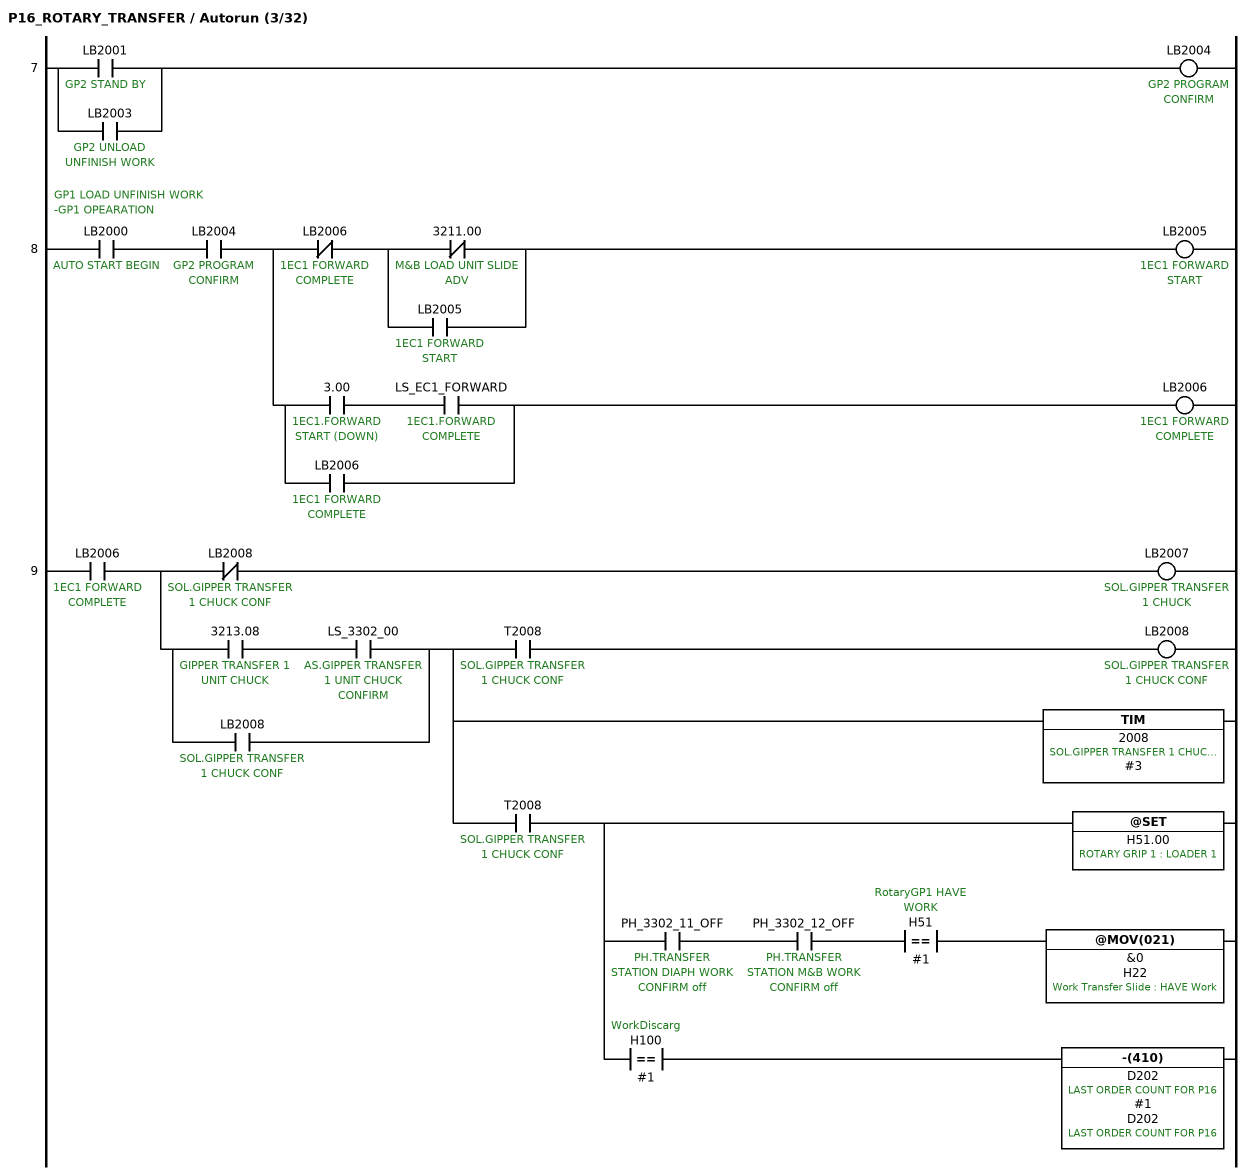
; [picture p240: P16_ROTARY_TRANSFER / Autorun, rungs 7-9]
; rung 7
LD LB2001  ; GP2 STAND BY
OR LB2003  ; GP2 UNLOAD UNFINISH WORK
OUT LB2004  ; GP2 PROGRAM CONFIRM
; rung 8: GP1 LOAD UNFINISH WORK / -GP1 OPEARATION
LD LB2000  ; AUTO START BEGIN
AND LB2004  ; GP2 PROGRAM CONFIRM
OUT TR0
ANDNOT LB2006  ; 1EC1 FORWARD COMPLETE
LDNOT 3211.00  ; M&B LOAD UNIT SLIDE ADV
OR LB2005  ; 1EC1 FORWARD START
ANDLD
OUT LB2005  ; 1EC1 FORWARD START
LD TR0
LD 3.00  ; 1EC1.FORWARD START (DOWN)
AND LS_EC1_FORWARD  ; 1EC1.FORWARD COMPLETE
OR LB2006  ; 1EC1 FORWARD COMPLETE
ANDLD
OUT LB2006  ; 1EC1 FORWARD COMPLETE
; rung 9
LD LB2006  ; 1EC1 FORWARD COMPLETE
OUT TR0
ANDNOT LB2008  ; SOL.GIPPER TRANSFER 1 CHUCK CONF
OUT LB2007  ; SOL.GIPPER TRANSFER 1 CHUCK
LD TR0
LD 3213.08  ; GIPPER TRANSFER 1 UNIT CHUCK
AND LS_3302_00  ; AS.GIPPER TRANSFER 1 UNIT CHUCK CONFIRM
OR LB2008  ; SOL.GIPPER TRANSFER 1 CHUCK CONF
ANDLD
OUT TR0
AND T2008  ; SOL.GIPPER TRANSFER 1 CHUCK CONF
OUT LB2008  ; SOL.GIPPER TRANSFER 1 CHUCK CONF
LD TR0
TIM 2008 #3  ; SOL.GIPPER TRANSFER 1 CHUCK CONF
AND T2008  ; SOL.GIPPER TRANSFER 1 CHUCK CONF
OUT TR0
@SET H51.00  ; ROTARY GRIP 1 : LOADER 1
AND PH_3302_11_OFF  ; PH.TRANSFER STATION DIAPH WORK CONFIRM off
AND PH_3302_12_OFF  ; PH.TRANSFER STATION M&B WORK CONFIRM off
AND=(300) H51 #1  ; RotaryGP1 HAVE WORK
@MOV(021) &0 H22  ; Work Transfer Slide : HAVE Work
LD TR0
AND=(300) H100 #1  ; WorkDiscarg
-(410) D202 #1 D202  ; LAST ORDER COUNT FOR P16

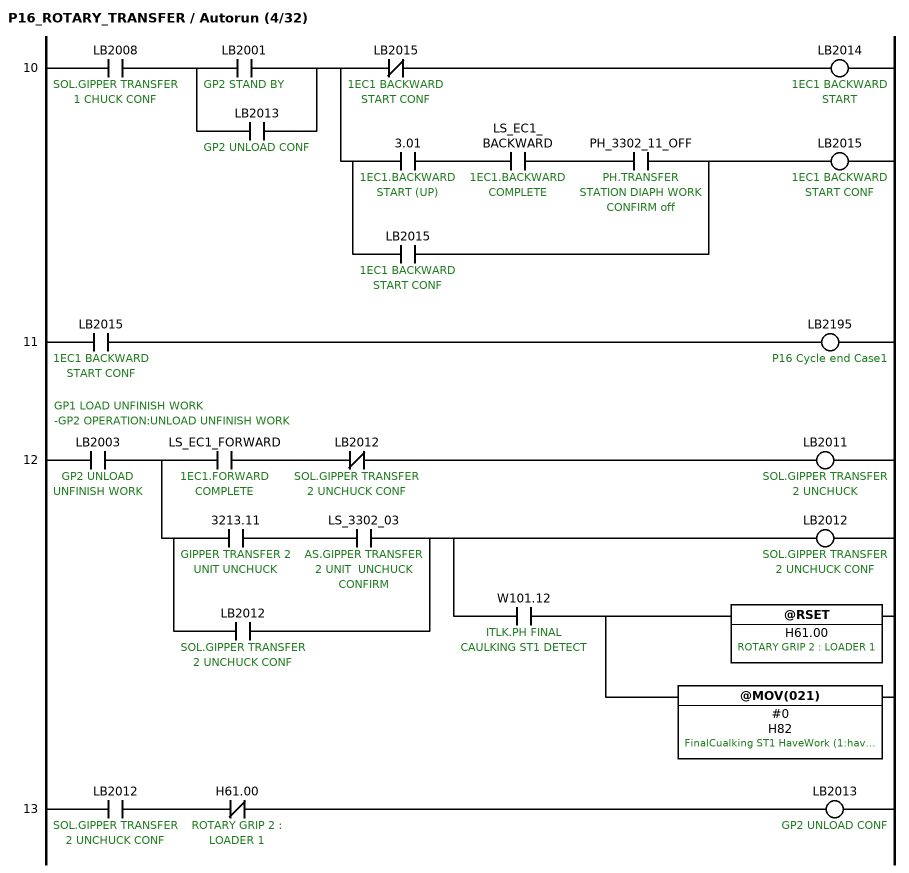
; rung 10
LD LB2008  ; SOL.GIPPER TRANSFER 1 CHUCK CONF
LD LB2001  ; GP2 STAND BY
OR LB2013  ; GP2 UNLOAD CONF
ANDLD
OUT TR0
ANDNOT LB2015  ; 1EC1 BACKWARD START CONF
OUT LB2014  ; 1EC1 BACKWARD START
LD TR0
LD 3.01  ; 1EC1.BACKWARD START (UP)
AND LS_EC1_BACKWARD  ; 1EC1.BACKWARD COMPLETE
AND PH_3302_11_OFF  ; PH.TRANSFER STATION DIAPH WORK CONFIRM off
OR LB2015  ; 1EC1 BACKWARD START CONF
ANDLD
OUT LB2015  ; 1EC1 BACKWARD START CONF
; rung 11
LD LB2015  ; 1EC1 BACKWARD START CONF
OUT LB2195  ; P16 Cycle end Case1
; rung 12: GP1 LOAD UNFINISH WORK / -GP2 OPERATION:UNLOAD UNFINISH WORK
LD LB2003  ; GP2 UNLOAD UNFINISH WORK
OUT TR0
AND LS_EC1_FORWARD  ; 1EC1.FORWARD COMPLETE
ANDNOT LB2012  ; SOL.GIPPER TRANSFER 2 UNCHUCK CONF
OUT LB2011  ; SOL.GIPPER TRANSFER 2 UNCHUCK
LD TR0
LD 3213.11  ; GIPPER TRANSFER 2 UNIT UNCHUCK
AND LS_3302_03  ; AS.GIPPER TRANSFER 2 UNIT  UNCHUCK CONFIRM
OR LB2012  ; SOL.GIPPER TRANSFER 2 UNCHUCK CONF
ANDLD
OUT LB2012  ; SOL.GIPPER TRANSFER 2 UNCHUCK CONF
AND W101.12  ; ITLK.PH FINAL CAULKING ST1 DETECT
@RSET H61.00  ; ROTARY GRIP 2 : LOADER 1
@MOV(021) #0 H82  ; FinalCualking ST1 HaveWork (1:have work 2:no work)
; rung 13
LD LB2012  ; SOL.GIPPER TRANSFER 2 UNCHUCK CONF
ANDNOT H61.00  ; ROTARY GRIP 2 : LOADER 1
OUT LB2013  ; GP2 UNLOAD CONF

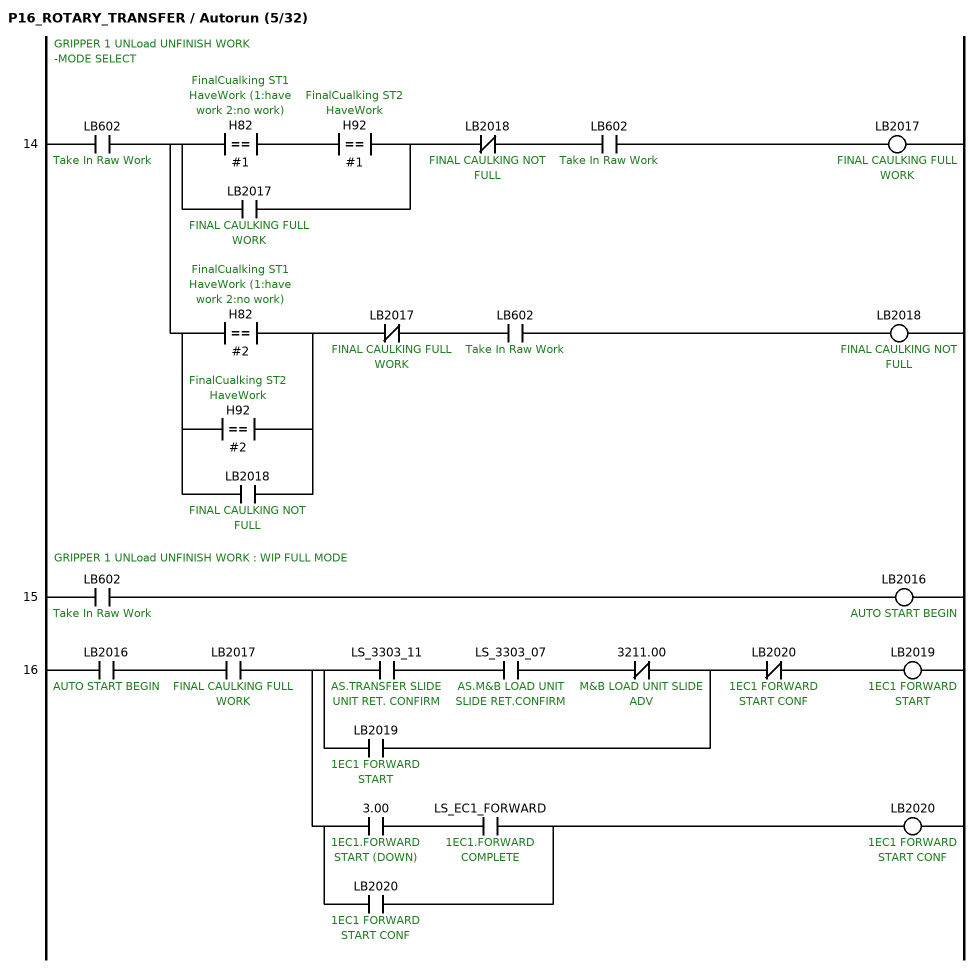
; rung 14: GRIPPER 1 UNLoad UNFINISH WORK / -MODE SELECT
LD LB602  ; Take In Raw Work
OUT TR0
LD=(300) H82 #1  ; FinalCualking ST1 HaveWork (1:have work 2:no work)
AND=(300) H92 #1  ; FinalCualking ST2 HaveWork
OR LB2017  ; FINAL CAULKING FULL WORK
ANDLD
ANDNOT LB2018  ; FINAL CAULKING NOT FULL
AND LB602  ; Take In Raw Work
OUT LB2017  ; FINAL CAULKING FULL WORK
LD TR0
LD=(300) H82 #2  ; FinalCualking ST1 HaveWork (1:have work 2:no work)
OR=(300) H92 #2  ; FinalCualking ST2 HaveWork
OR LB2018  ; FINAL CAULKING NOT FULL
ANDLD
ANDNOT LB2017  ; FINAL CAULKING FULL WORK
AND LB602  ; Take In Raw Work
OUT LB2018  ; FINAL CAULKING NOT FULL
; rung 15: GRIPPER 1 UNLoad UNFINISH WORK : WIP FULL MODE
LD LB602  ; Take In Raw Work
OUT LB2016  ; AUTO START BEGIN
; rung 16
LD LB2016  ; AUTO START BEGIN
AND LB2017  ; FINAL CAULKING FULL WORK
OUT TR0
LD LS_3303_11  ; AS.TRANSFER SLIDE UNIT RET. CONFIRM
AND LS_3303_07  ; AS.M&B LOAD UNIT SLIDE RET.CONFIRM
ANDNOT 3211.00  ; M&B LOAD UNIT SLIDE ADV
OR LB2019  ; 1EC1 FORWARD START
ANDLD
ANDNOT LB2020  ; 1EC1 FORWARD START CONF
OUT LB2019  ; 1EC1 FORWARD START
LD TR0
LD 3.00  ; 1EC1.FORWARD START (DOWN)
AND LS_EC1_FORWARD  ; 1EC1.FORWARD COMPLETE
OR LB2020  ; 1EC1 FORWARD START CONF
ANDLD
OUT LB2020  ; 1EC1 FORWARD START CONF

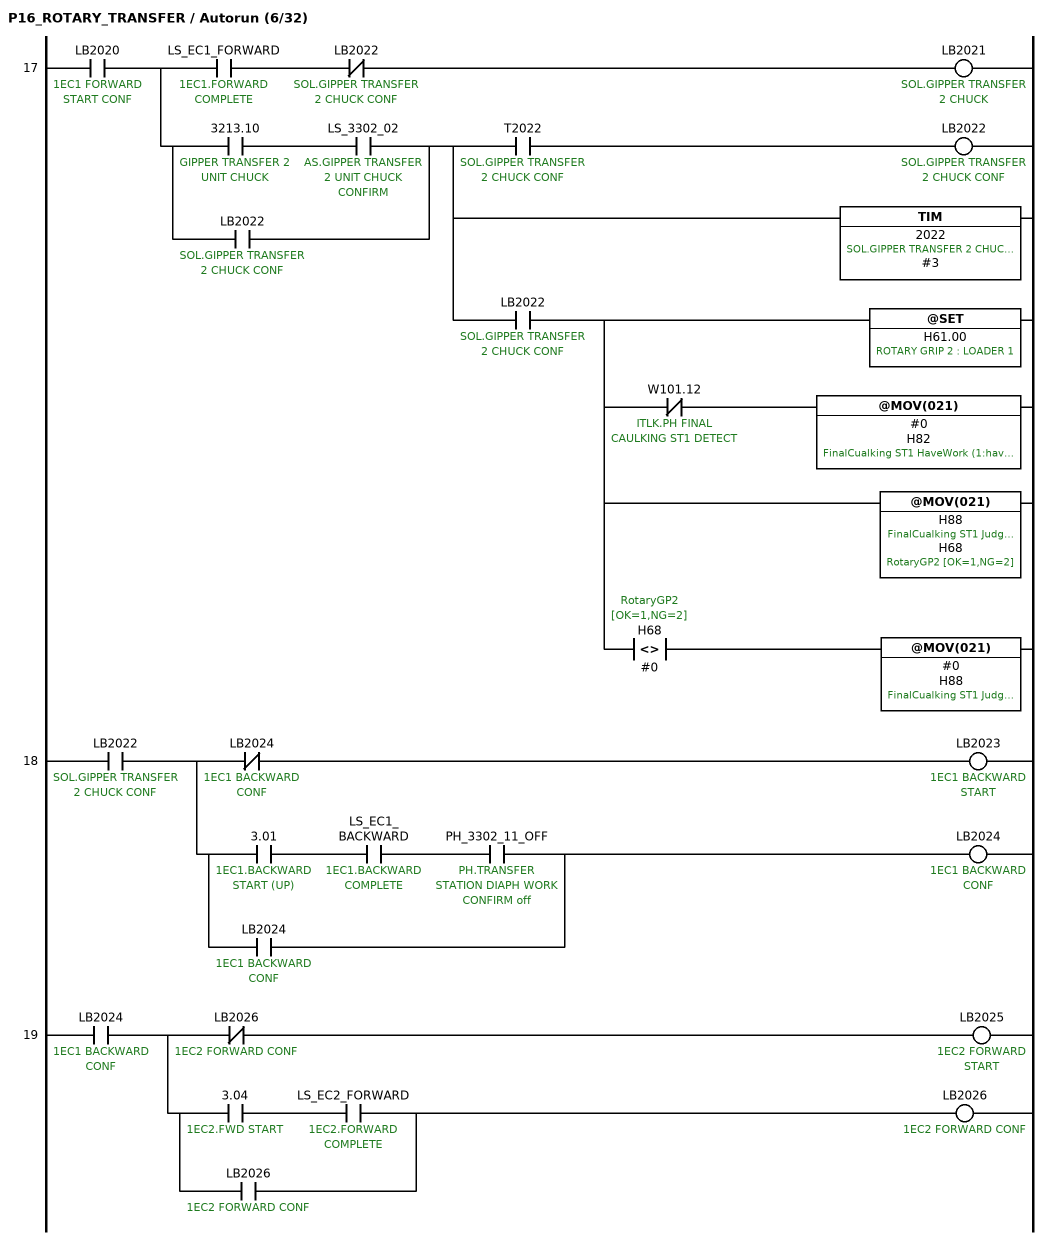
; rung 17
LD LB2020  ; 1EC1 FORWARD START CONF
OUT TR0
AND LS_EC1_FORWARD  ; 1EC1.FORWARD COMPLETE
ANDNOT LB2022  ; SOL.GIPPER TRANSFER 2 CHUCK CONF
OUT LB2021  ; SOL.GIPPER TRANSFER 2 CHUCK
LD TR0
LD 3213.10  ; GIPPER TRANSFER 2 UNIT CHUCK
AND LS_3302_02  ; AS.GIPPER TRANSFER 2 UNIT CHUCK CONFIRM
OR LB2022  ; SOL.GIPPER TRANSFER 2 CHUCK CONF
ANDLD
OUT TR0
AND T2022  ; SOL.GIPPER TRANSFER 2 CHUCK CONF
OUT LB2022  ; SOL.GIPPER TRANSFER 2 CHUCK CONF
LD TR0
TIM 2022 #3  ; SOL.GIPPER TRANSFER 2 CHUCK CONF
AND LB2022  ; SOL.GIPPER TRANSFER 2 CHUCK CONF
OUT TR0
@SET H61.00  ; ROTARY GRIP 2 : LOADER 1
ANDNOT W101.12  ; ITLK.PH FINAL CAULKING ST1 DETECT
@MOV(021) #0 H82  ; FinalCualking ST1 HaveWork (1:have work 2:no work)
LD TR0
@MOV(021) H88 H68  ; FinalCualking ST1 Judge [OK=1,NG=2], RotaryGP2 [OK=1,NG=2]
AND<>(305) H68 #0  ; RotaryGP2 [OK=1,NG=2]
@MOV(021) #0 H88  ; FinalCualking ST1 Judge [OK=1,NG=2]
; rung 18
LD LB2022  ; SOL.GIPPER TRANSFER 2 CHUCK CONF
OUT TR0
ANDNOT LB2024  ; 1EC1 BACKWARD CONF
OUT LB2023  ; 1EC1 BACKWARD START
LD TR0
LD 3.01  ; 1EC1.BACKWARD START (UP)
AND LS_EC1_BACKWARD  ; 1EC1.BACKWARD COMPLETE
AND PH_3302_11_OFF  ; PH.TRANSFER STATION DIAPH WORK CONFIRM off
OR LB2024  ; 1EC1 BACKWARD CONF
ANDLD
OUT LB2024  ; 1EC1 BACKWARD CONF
; rung 19
LD LB2024  ; 1EC1 BACKWARD CONF
OUT TR0
ANDNOT LB2026  ; 1EC2 FORWARD CONF
OUT LB2025  ; 1EC2 FORWARD START
LD TR0
LD 3.04  ; 1EC2.FWD START
AND LS_EC2_FORWARD  ; 1EC2.FORWARD COMPLETE
OR LB2026  ; 1EC2 FORWARD CONF
ANDLD
OUT LB2026  ; 1EC2 FORWARD CONF

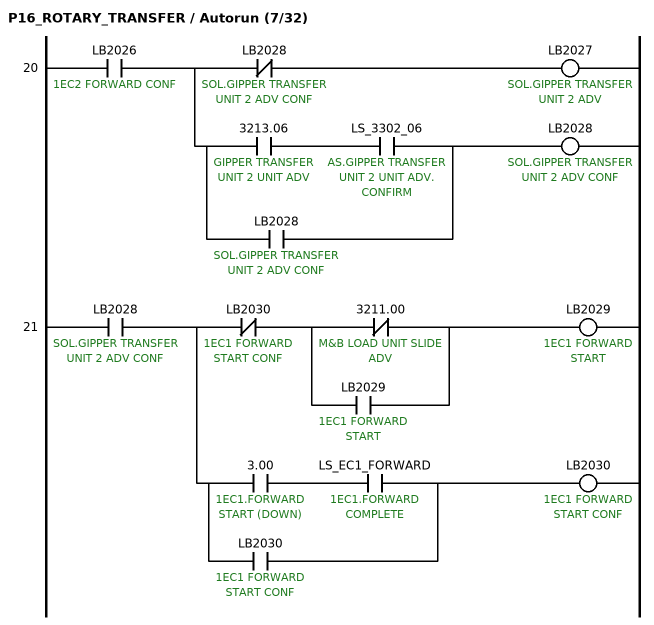
; rung 20
LD LB2026  ; 1EC2 FORWARD CONF
OUT TR0
ANDNOT LB2028  ; SOL.GIPPER TRANSFER UNIT 2 ADV CONF
OUT LB2027  ; SOL.GIPPER TRANSFER UNIT 2 ADV
LD TR0
LD 3213.06  ; GIPPER TRANSFER UNIT 2 UNIT ADV
AND LS_3302_06  ; AS.GIPPER TRANSFER UNIT 2 UNIT ADV. CONFIRM
OR LB2028  ; SOL.GIPPER TRANSFER UNIT 2 ADV CONF
ANDLD
OUT LB2028  ; SOL.GIPPER TRANSFER UNIT 2 ADV CONF
; rung 21
LD LB2028  ; SOL.GIPPER TRANSFER UNIT 2 ADV CONF
OUT TR0
ANDNOT LB2030  ; 1EC1 FORWARD START CONF
LDNOT 3211.00  ; M&B LOAD UNIT SLIDE ADV
OR LB2029  ; 1EC1 FORWARD START
ANDLD
OUT LB2029  ; 1EC1 FORWARD START
LD TR0
LD 3.00  ; 1EC1.FORWARD START (DOWN)
AND LS_EC1_FORWARD  ; 1EC1.FORWARD COMPLETE
OR LB2030  ; 1EC1 FORWARD START CONF
ANDLD
OUT LB2030  ; 1EC1 FORWARD START CONF

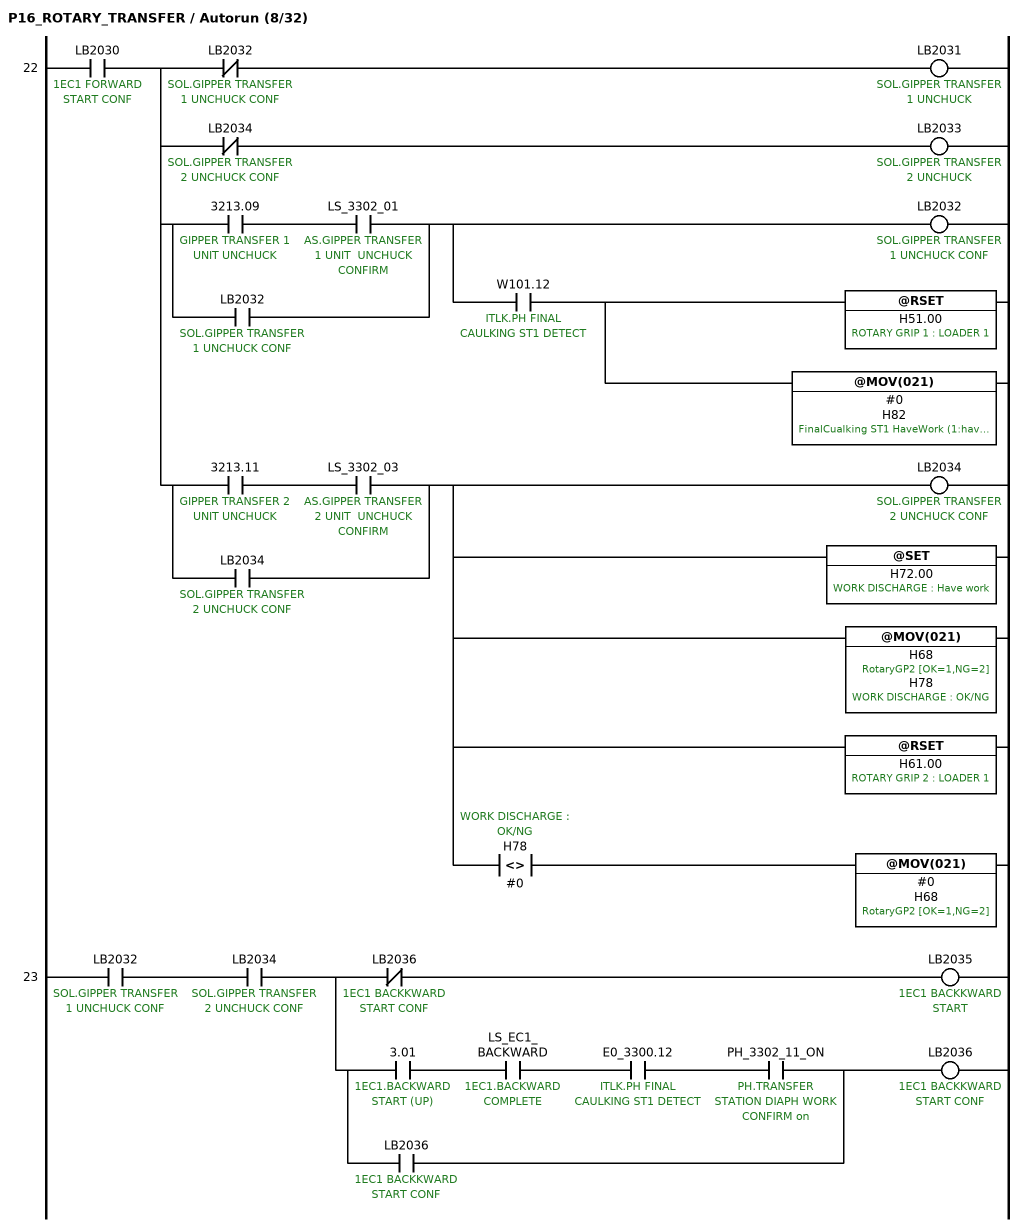
; rung 22
LD LB2030  ; 1EC1 FORWARD START CONF
OUT TR0
ANDNOT LB2032  ; SOL.GIPPER TRANSFER 1 UNCHUCK CONF
OUT LB2031  ; SOL.GIPPER TRANSFER 1 UNCHUCK
LD TR0
ANDNOT LB2034  ; SOL.GIPPER TRANSFER 2 UNCHUCK CONF
OUT LB2033  ; SOL.GIPPER TRANSFER 2 UNCHUCK
LD TR0
LD 3213.09  ; GIPPER TRANSFER 1 UNIT UNCHUCK
AND LS_3302_01  ; AS.GIPPER TRANSFER 1 UNIT  UNCHUCK CONFIRM
OR LB2032  ; SOL.GIPPER TRANSFER 1 UNCHUCK CONF
ANDLD
OUT LB2032  ; SOL.GIPPER TRANSFER 1 UNCHUCK CONF
AND W101.12  ; ITLK.PH FINAL CAULKING ST1 DETECT
@RSET H51.00  ; ROTARY GRIP 1 : LOADER 1
@MOV(021) #0 H82  ; FinalCualking ST1 HaveWork (1:have work 2:no work)
LD TR0
LD 3213.11  ; GIPPER TRANSFER 2 UNIT UNCHUCK
AND LS_3302_03  ; AS.GIPPER TRANSFER 2 UNIT  UNCHUCK CONFIRM
OR LB2034  ; SOL.GIPPER TRANSFER 2 UNCHUCK CONF
ANDLD
OUT LB2034  ; SOL.GIPPER TRANSFER 2 UNCHUCK CONF
@SET H72.00  ; WORK DISCHARGE : Have work
@MOV(021) H68 H78  ; RotaryGP2 [OK=1,NG=2], WORK DISCHARGE : OK/NG
@RSET H61.00  ; ROTARY GRIP 2 : LOADER 1
AND<>(305) H78 #0  ; WORK DISCHARGE : OK/NG
@MOV(021) #0 H68  ; RotaryGP2 [OK=1,NG=2]
; rung 23
LD LB2032  ; SOL.GIPPER TRANSFER 1 UNCHUCK CONF
AND LB2034  ; SOL.GIPPER TRANSFER 2 UNCHUCK CONF
OUT TR0
ANDNOT LB2036  ; 1EC1 BACKKWARD START CONF
OUT LB2035  ; 1EC1 BACKKWARD START
LD TR0
LD 3.01  ; 1EC1.BACKWARD START (UP)
AND LS_EC1_BACKWARD  ; 1EC1.BACKWARD COMPLETE
AND E0_3300.12  ; ITLK.PH FINAL CAULKING ST1 DETECT
AND PH_3302_11_ON  ; PH.TRANSFER STATION DIAPH WORK CONFIRM on
OR LB2036  ; 1EC1 BACKKWARD START CONF
ANDLD
OUT LB2036  ; 1EC1 BACKKWARD START CONF

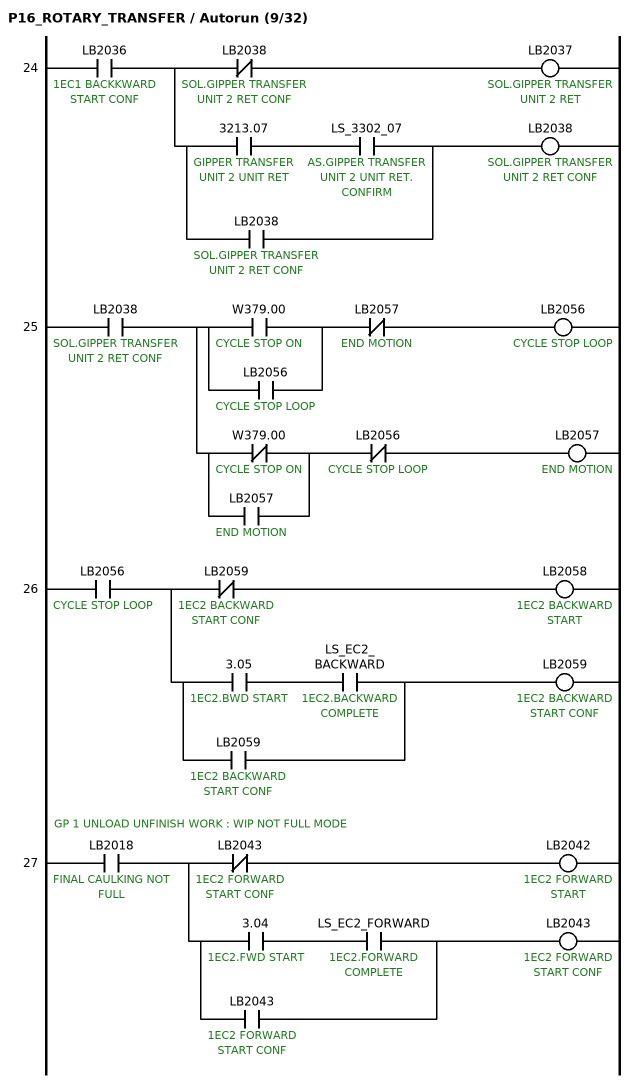
; rung 24
LD LB2036  ; 1EC1 BACKKWARD START CONF
OUT TR0
ANDNOT LB2038  ; SOL.GIPPER TRANSFER UNIT 2 RET CONF
OUT LB2037  ; SOL.GIPPER TRANSFER UNIT 2 RET
LD TR0
LD 3213.07  ; GIPPER TRANSFER UNIT 2 UNIT RET
AND LS_3302_07  ; AS.GIPPER TRANSFER UNIT 2 UNIT RET. CONFIRM
OR LB2038  ; SOL.GIPPER TRANSFER UNIT 2 RET CONF
ANDLD
OUT LB2038  ; SOL.GIPPER TRANSFER UNIT 2 RET CONF
; rung 25
LD LB2038  ; SOL.GIPPER TRANSFER UNIT 2 RET CONF
OUT TR0
LD W379.00  ; CYCLE STOP ON
OR LB2056  ; CYCLE STOP LOOP
ANDLD
ANDNOT LB2057  ; END MOTION
OUT LB2056  ; CYCLE STOP LOOP
LD TR0
LDNOT W379.00  ; CYCLE STOP ON
OR LB2057  ; END MOTION
ANDLD
ANDNOT LB2056  ; CYCLE STOP LOOP
OUT LB2057  ; END MOTION
; rung 26
LD LB2056  ; CYCLE STOP LOOP
OUT TR0
ANDNOT LB2059  ; 1EC2 BACKWARD START CONF
OUT LB2058  ; 1EC2 BACKWARD START
LD TR0
LD 3.05  ; 1EC2.BWD START
AND LS_EC2_BACKWARD  ; 1EC2.BACKWARD COMPLETE
OR LB2059  ; 1EC2 BACKWARD START CONF
ANDLD
OUT LB2059  ; 1EC2 BACKWARD START CONF
; rung 27: GP 1 UNLOAD UNFINISH WORK : WIP NOT FULL MODE
LD LB2018  ; FINAL CAULKING NOT FULL
OUT TR0
ANDNOT LB2043  ; 1EC2 FORWARD START CONF
OUT LB2042  ; 1EC2 FORWARD START
LD TR0
LD 3.04  ; 1EC2.FWD START
AND LS_EC2_FORWARD  ; 1EC2.FORWARD COMPLETE
OR LB2043  ; 1EC2 FORWARD START CONF
ANDLD
OUT LB2043  ; 1EC2 FORWARD START CONF

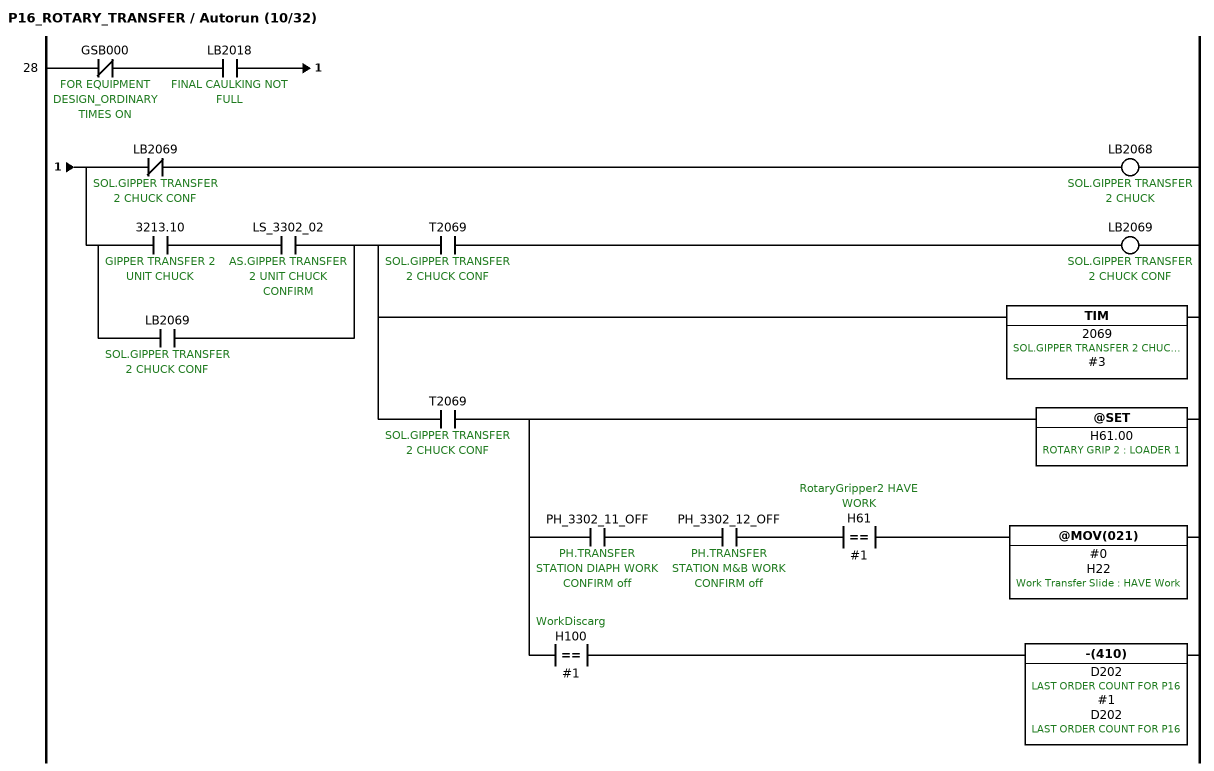
; rung 28
LDNOT GSB000  ; FOR EQUIPMENT DESIGN_ORDINARY TIMES ON
AND LB2018  ; FINAL CAULKING NOT FULL
OUT TR0
ANDNOT LB2069  ; SOL.GIPPER TRANSFER 2 CHUCK CONF
OUT LB2068  ; SOL.GIPPER TRANSFER 2 CHUCK
LD TR0
LD 3213.10  ; GIPPER TRANSFER 2 UNIT CHUCK
AND LS_3302_02  ; AS.GIPPER TRANSFER 2 UNIT CHUCK CONFIRM
OR LB2069  ; SOL.GIPPER TRANSFER 2 CHUCK CONF
ANDLD
OUT TR0
AND T2069  ; SOL.GIPPER TRANSFER 2 CHUCK CONF
OUT LB2069  ; SOL.GIPPER TRANSFER 2 CHUCK CONF
LD TR0
TIM 2069 #3  ; SOL.GIPPER TRANSFER 2 CHUCK CONF
AND T2069  ; SOL.GIPPER TRANSFER 2 CHUCK CONF
OUT TR0
@SET H61.00  ; ROTARY GRIP 2 : LOADER 1
AND PH_3302_11_OFF  ; PH.TRANSFER STATION DIAPH WORK CONFIRM off
AND PH_3302_12_OFF  ; PH.TRANSFER STATION M&B WORK CONFIRM off
AND=(300) H61 #1  ; RotaryGripper2 HAVE WORK
@MOV(021) #0 H22  ; Work Transfer Slide : HAVE Work
LD TR0
AND=(300) H100 #1  ; WorkDiscarg
-(410) D202 #1 D202  ; LAST ORDER COUNT FOR P16

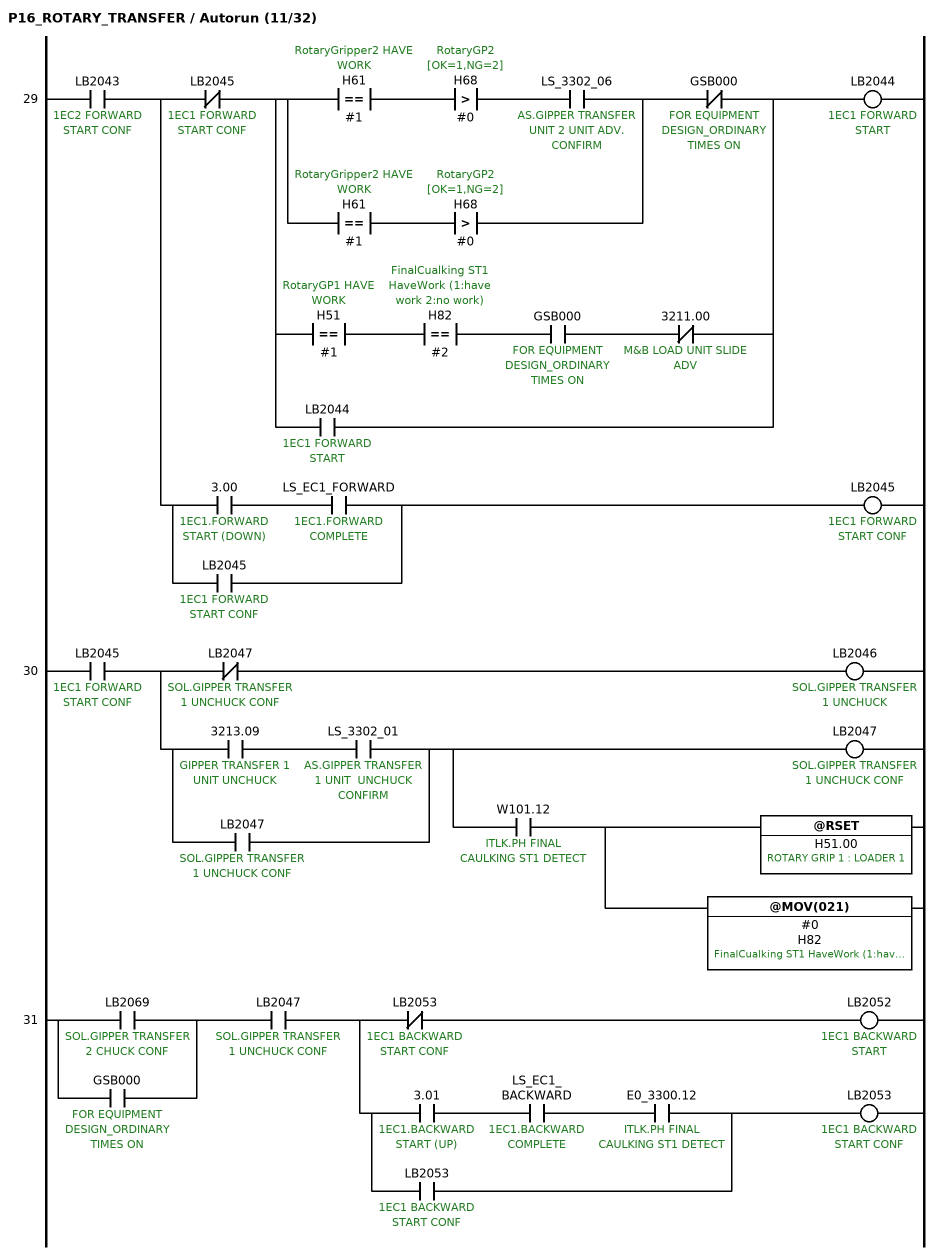
; rung 29
LD LB2043  ; 1EC2 FORWARD START CONF
OUT TR0
ANDNOT LB2045  ; 1EC1 FORWARD START CONF
LD=(300) H61 #1  ; RotaryGripper2 HAVE WORK
AND>(320) H68 #0  ; RotaryGP2 [OK=1,NG=2]
AND LS_3302_06  ; AS.GIPPER TRANSFER UNIT 2 UNIT ADV. CONFIRM
LD=(300) H61 #1  ; RotaryGripper2 HAVE WORK
AND>(320) H68 #0  ; RotaryGP2 [OK=1,NG=2]
ORLD
ANDNOT GSB000  ; FOR EQUIPMENT DESIGN_ORDINARY TIMES ON
LD=(300) H51 #1  ; RotaryGP1 HAVE WORK
AND=(300) H82 #2  ; FinalCualking ST1 HaveWork (1:have work 2:no work)
AND GSB000  ; FOR EQUIPMENT DESIGN_ORDINARY TIMES ON
ANDNOT 3211.00  ; M&B LOAD UNIT SLIDE ADV
ORLD
OR LB2044  ; 1EC1 FORWARD START
ANDLD
OUT LB2044  ; 1EC1 FORWARD START
LD TR0
LD 3.00  ; 1EC1.FORWARD START (DOWN)
AND LS_EC1_FORWARD  ; 1EC1.FORWARD COMPLETE
OR LB2045  ; 1EC1 FORWARD START CONF
ANDLD
OUT LB2045  ; 1EC1 FORWARD START CONF
; rung 30
LD LB2045  ; 1EC1 FORWARD START CONF
OUT TR0
ANDNOT LB2047  ; SOL.GIPPER TRANSFER 1 UNCHUCK CONF
OUT LB2046  ; SOL.GIPPER TRANSFER 1 UNCHUCK
LD TR0
LD 3213.09  ; GIPPER TRANSFER 1 UNIT UNCHUCK
AND LS_3302_01  ; AS.GIPPER TRANSFER 1 UNIT  UNCHUCK CONFIRM
OR LB2047  ; SOL.GIPPER TRANSFER 1 UNCHUCK CONF
ANDLD
OUT LB2047  ; SOL.GIPPER TRANSFER 1 UNCHUCK CONF
AND W101.12  ; ITLK.PH FINAL CAULKING ST1 DETECT
@RSET H51.00  ; ROTARY GRIP 1 : LOADER 1
@MOV(021) #0 H82  ; FinalCualking ST1 HaveWork (1:have work 2:no work)
; rung 31
LD LB2069  ; SOL.GIPPER TRANSFER 2 CHUCK CONF
OR GSB000  ; FOR EQUIPMENT DESIGN_ORDINARY TIMES ON
AND LB2047  ; SOL.GIPPER TRANSFER 1 UNCHUCK CONF
OUT TR0
ANDNOT LB2053  ; 1EC1 BACKWARD START CONF
OUT LB2052  ; 1EC1 BACKWARD START
LD TR0
LD 3.01  ; 1EC1.BACKWARD START (UP)
AND LS_EC1_BACKWARD  ; 1EC1.BACKWARD COMPLETE
AND E0_3300.12  ; ITLK.PH FINAL CAULKING ST1 DETECT
OR LB2053  ; 1EC1 BACKWARD START CONF
ANDLD
OUT LB2053  ; 1EC1 BACKWARD START CONF

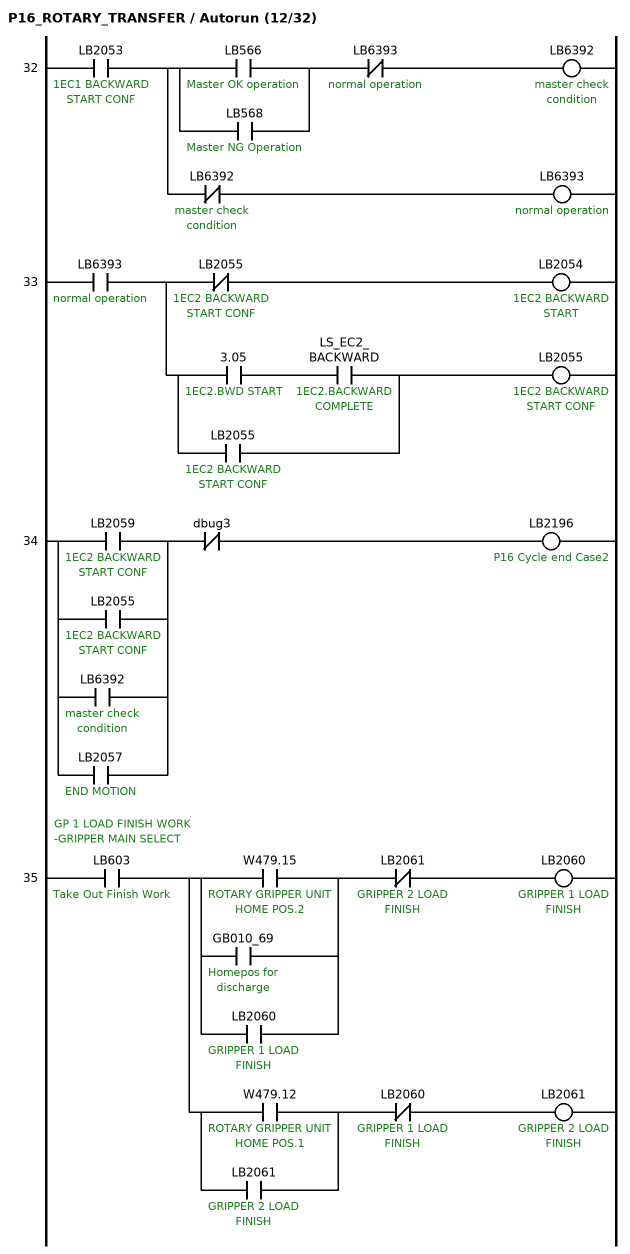
; rung 32
LD LB2053  ; 1EC1 BACKWARD START CONF
OUT TR0
LD LB566  ; Master OK operation
OR LB568  ; Master NG Operation
ANDLD
ANDNOT LB6393  ; normal operation
OUT LB6392  ; master check condition
LD TR0
ANDNOT LB6392  ; master check condition
OUT LB6393  ; normal operation
; rung 33
LD LB6393  ; normal operation
OUT TR0
ANDNOT LB2055  ; 1EC2 BACKWARD START CONF
OUT LB2054  ; 1EC2 BACKWARD START
LD TR0
LD 3.05  ; 1EC2.BWD START
AND LS_EC2_BACKWARD  ; 1EC2.BACKWARD COMPLETE
OR LB2055  ; 1EC2 BACKWARD START CONF
ANDLD
OUT LB2055  ; 1EC2 BACKWARD START CONF
; rung 34
LD LB2059  ; 1EC2 BACKWARD START CONF
OR LB2055  ; 1EC2 BACKWARD START CONF
OR LB6392  ; master check condition
OR LB2057  ; END MOTION
ANDNOT dbug3
OUT LB2196  ; P16 Cycle end Case2
; rung 35: GP 1 LOAD FINISH WORK / -GRIPPER MAIN SELECT
LD LB603  ; Take Out Finish Work
OUT TR0
LD W479.15  ; ROTARY GRIPPER UNIT HOME POS.2
OR GB010_69  ; Homepos for discharge
OR LB2060  ; GRIPPER 1 LOAD FINISH
ANDLD
ANDNOT LB2061  ; GRIPPER 2 LOAD FINISH
OUT LB2060  ; GRIPPER 1 LOAD FINISH
LD TR0
LD W479.12  ; ROTARY GRIPPER UNIT HOME POS.1
OR LB2061  ; GRIPPER 2 LOAD FINISH
ANDLD
ANDNOT LB2060  ; GRIPPER 1 LOAD FINISH
OUT LB2061  ; GRIPPER 2 LOAD FINISH

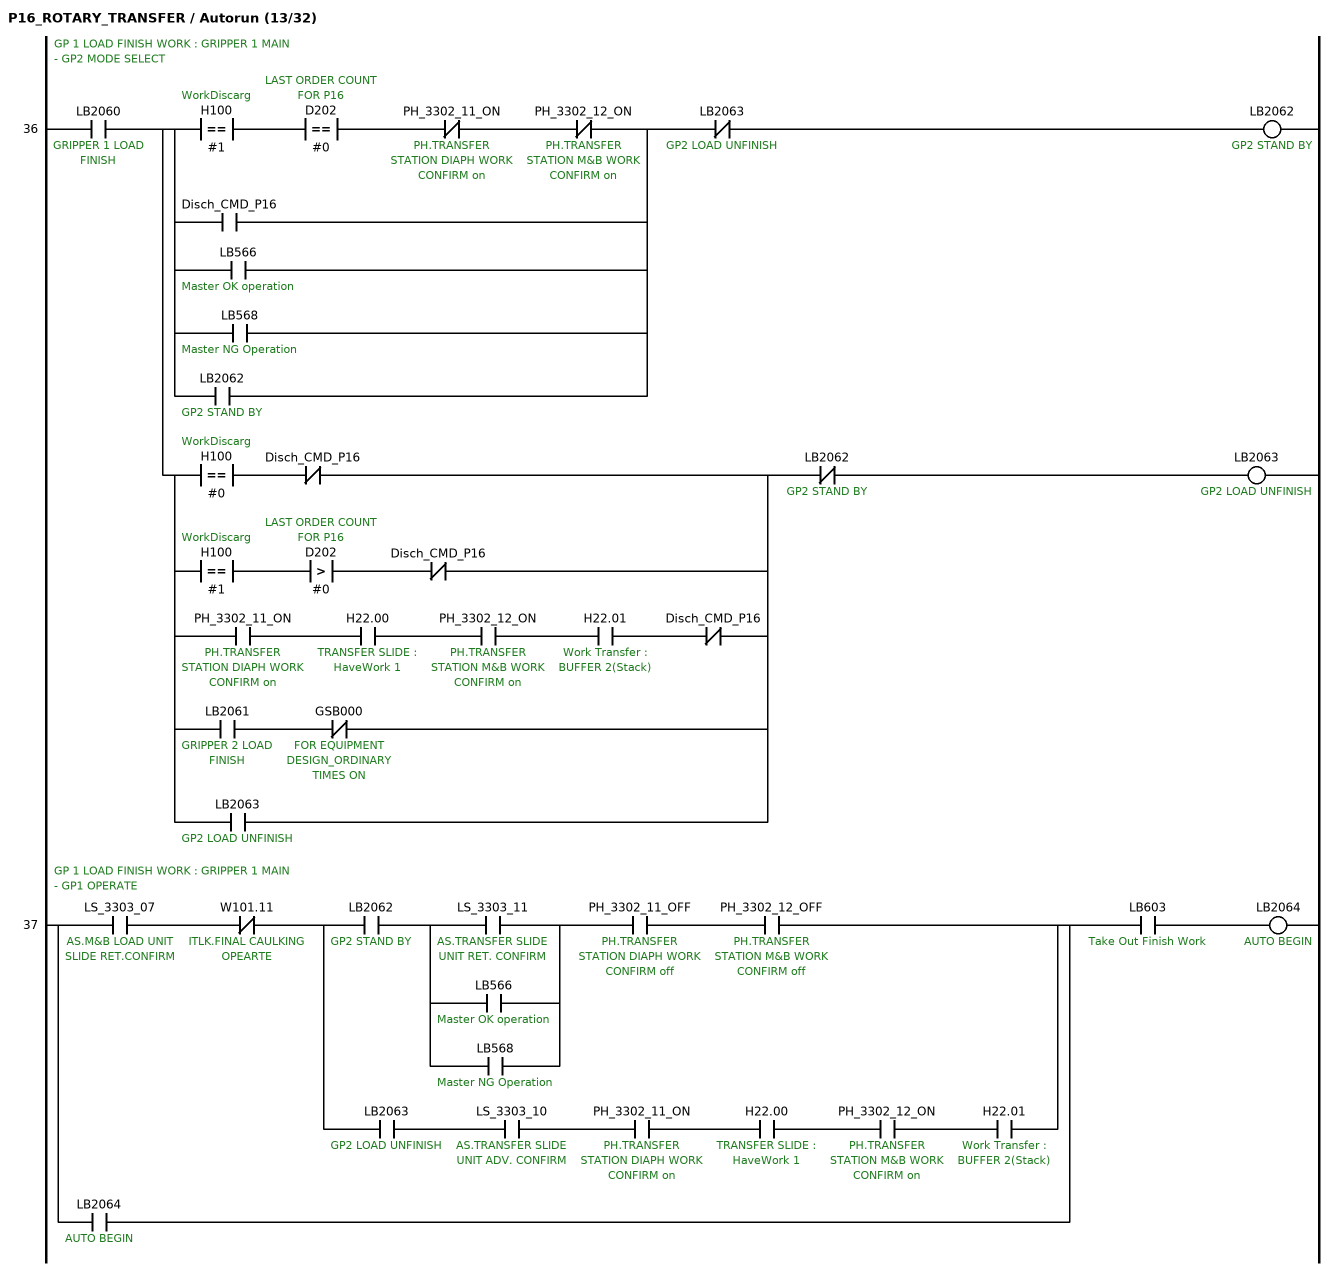
; rung 36: GP 1 LOAD FINISH WORK : GRIPPER 1 MAIN / - GP2 MODE SELECT
LD LB2060  ; GRIPPER 1 LOAD FINISH
OUT TR0
LD=(300) H100 #1  ; WorkDiscarg
AND=(300) D202 #0  ; LAST ORDER COUNT FOR P16
ANDNOT PH_3302_11_ON  ; PH.TRANSFER STATION DIAPH WORK CONFIRM on
ANDNOT PH_3302_12_ON  ; PH.TRANSFER STATION M&B WORK CONFIRM on
OR Disch_CMD_P16
OR LB566  ; Master OK operation
OR LB568  ; Master NG Operation
OR LB2062  ; GP2 STAND BY
ANDLD
ANDNOT LB2063  ; GP2 LOAD UNFINISH
OUT LB2062  ; GP2 STAND BY
LD TR0
LD=(300) H100 #0  ; WorkDiscarg
ANDNOT Disch_CMD_P16
LD=(300) H100 #1  ; WorkDiscarg
AND>(320) D202 #0  ; LAST ORDER COUNT FOR P16
ANDNOT Disch_CMD_P16
ORLD
LD PH_3302_11_ON  ; PH.TRANSFER STATION DIAPH WORK CONFIRM on
AND H22.00  ; TRANSFER SLIDE : HaveWork 1
AND PH_3302_12_ON  ; PH.TRANSFER STATION M&B WORK CONFIRM on
AND H22.01  ; Work Transfer : BUFFER 2(Stack)
ANDNOT Disch_CMD_P16
ORLD
LD LB2061  ; GRIPPER 2 LOAD FINISH
ANDNOT GSB000  ; FOR EQUIPMENT DESIGN_ORDINARY TIMES ON
ORLD
OR LB2063  ; GP2 LOAD UNFINISH
ANDLD
ANDNOT LB2062  ; GP2 STAND BY
OUT LB2063  ; GP2 LOAD UNFINISH
; rung 37: GP 1 LOAD FINISH WORK : GRIPPER 1 MAIN / - GP1 OPERATE
LD LS_3303_07  ; AS.M&B LOAD UNIT SLIDE RET.CONFIRM
ANDNOT W101.11  ; ITLK.FINAL CAULKING OPEARTE
LD LB2062  ; GP2 STAND BY
LD LS_3303_11  ; AS.TRANSFER SLIDE UNIT RET. CONFIRM
OR LB566  ; Master OK operation
OR LB568  ; Master NG Operation
ANDLD
AND PH_3302_11_OFF  ; PH.TRANSFER STATION DIAPH WORK CONFIRM off
AND PH_3302_12_OFF  ; PH.TRANSFER STATION M&B WORK CONFIRM off
LD LB2063  ; GP2 LOAD UNFINISH
AND LS_3303_10  ; AS.TRANSFER SLIDE UNIT ADV. CONFIRM
AND PH_3302_11_ON  ; PH.TRANSFER STATION DIAPH WORK CONFIRM on
AND H22.00  ; TRANSFER SLIDE : HaveWork 1
AND PH_3302_12_ON  ; PH.TRANSFER STATION M&B WORK CONFIRM on
AND H22.01  ; Work Transfer : BUFFER 2(Stack)
ORLD
ANDLD
OR LB2064  ; AUTO BEGIN
AND LB603  ; Take Out Finish Work
OUT LB2064  ; AUTO BEGIN

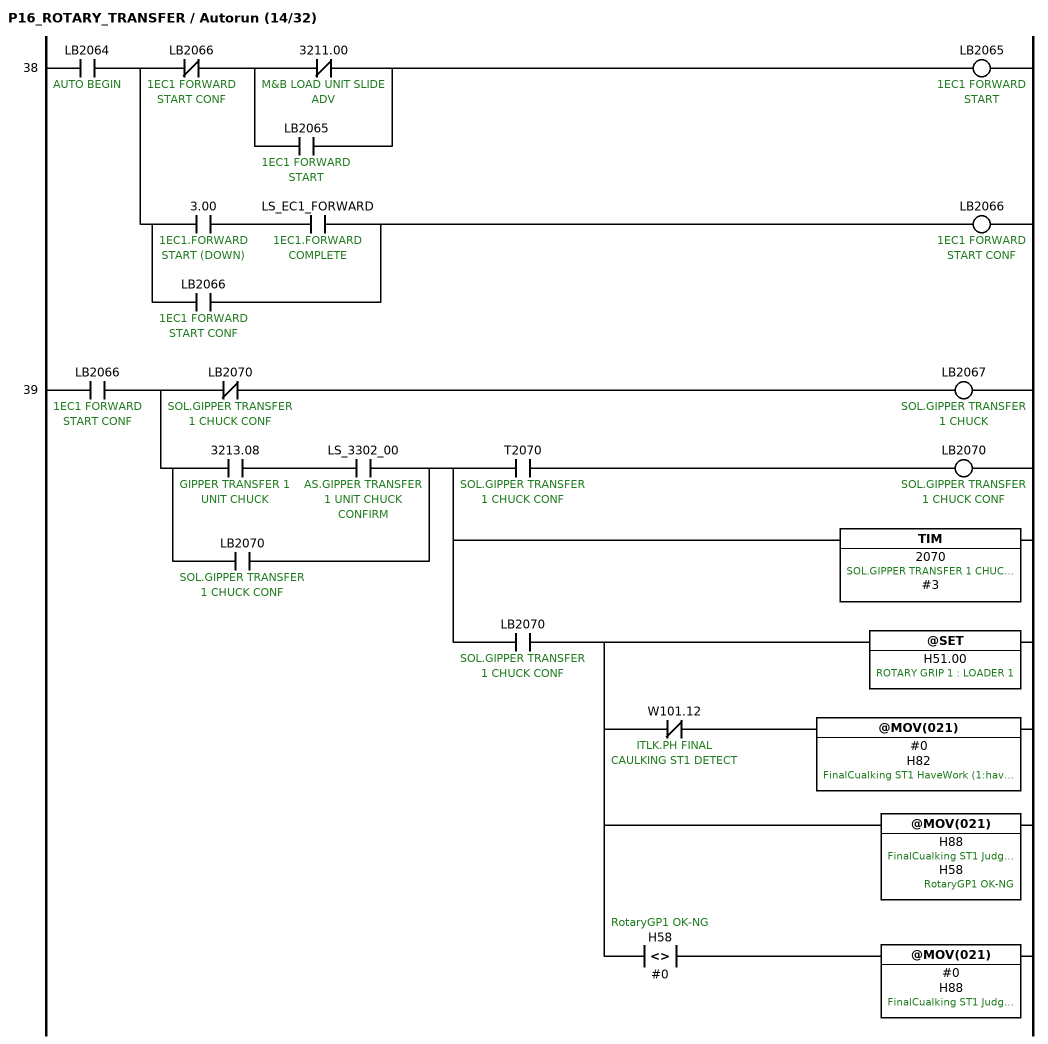
; rung 38
LD LB2064  ; AUTO BEGIN
OUT TR0
ANDNOT LB2066  ; 1EC1 FORWARD START CONF
LDNOT 3211.00  ; M&B LOAD UNIT SLIDE ADV
OR LB2065  ; 1EC1 FORWARD START
ANDLD
OUT LB2065  ; 1EC1 FORWARD START
LD TR0
LD 3.00  ; 1EC1.FORWARD START (DOWN)
AND LS_EC1_FORWARD  ; 1EC1.FORWARD COMPLETE
OR LB2066  ; 1EC1 FORWARD START CONF
ANDLD
OUT LB2066  ; 1EC1 FORWARD START CONF
; rung 39
LD LB2066  ; 1EC1 FORWARD START CONF
OUT TR0
ANDNOT LB2070  ; SOL.GIPPER TRANSFER 1 CHUCK CONF
OUT LB2067  ; SOL.GIPPER TRANSFER 1 CHUCK
LD TR0
LD 3213.08  ; GIPPER TRANSFER 1 UNIT CHUCK
AND LS_3302_00  ; AS.GIPPER TRANSFER 1 UNIT CHUCK CONFIRM
OR LB2070  ; SOL.GIPPER TRANSFER 1 CHUCK CONF
ANDLD
OUT TR0
AND T2070  ; SOL.GIPPER TRANSFER 1 CHUCK CONF
OUT LB2070  ; SOL.GIPPER TRANSFER 1 CHUCK CONF
LD TR0
TIM 2070 #3  ; SOL.GIPPER TRANSFER 1 CHUCK CONF
AND LB2070  ; SOL.GIPPER TRANSFER 1 CHUCK CONF
OUT TR0
@SET H51.00  ; ROTARY GRIP 1 : LOADER 1
ANDNOT W101.12  ; ITLK.PH FINAL CAULKING ST1 DETECT
@MOV(021) #0 H82  ; FinalCualking ST1 HaveWork (1:have work 2:no work)
LD TR0
@MOV(021) H88 H58  ; FinalCualking ST1 Judge [OK=1,NG=2], RotaryGP1 OK-NG
AND<>(305) H58 #0  ; RotaryGP1 OK-NG
@MOV(021) #0 H88  ; FinalCualking ST1 Judge [OK=1,NG=2]

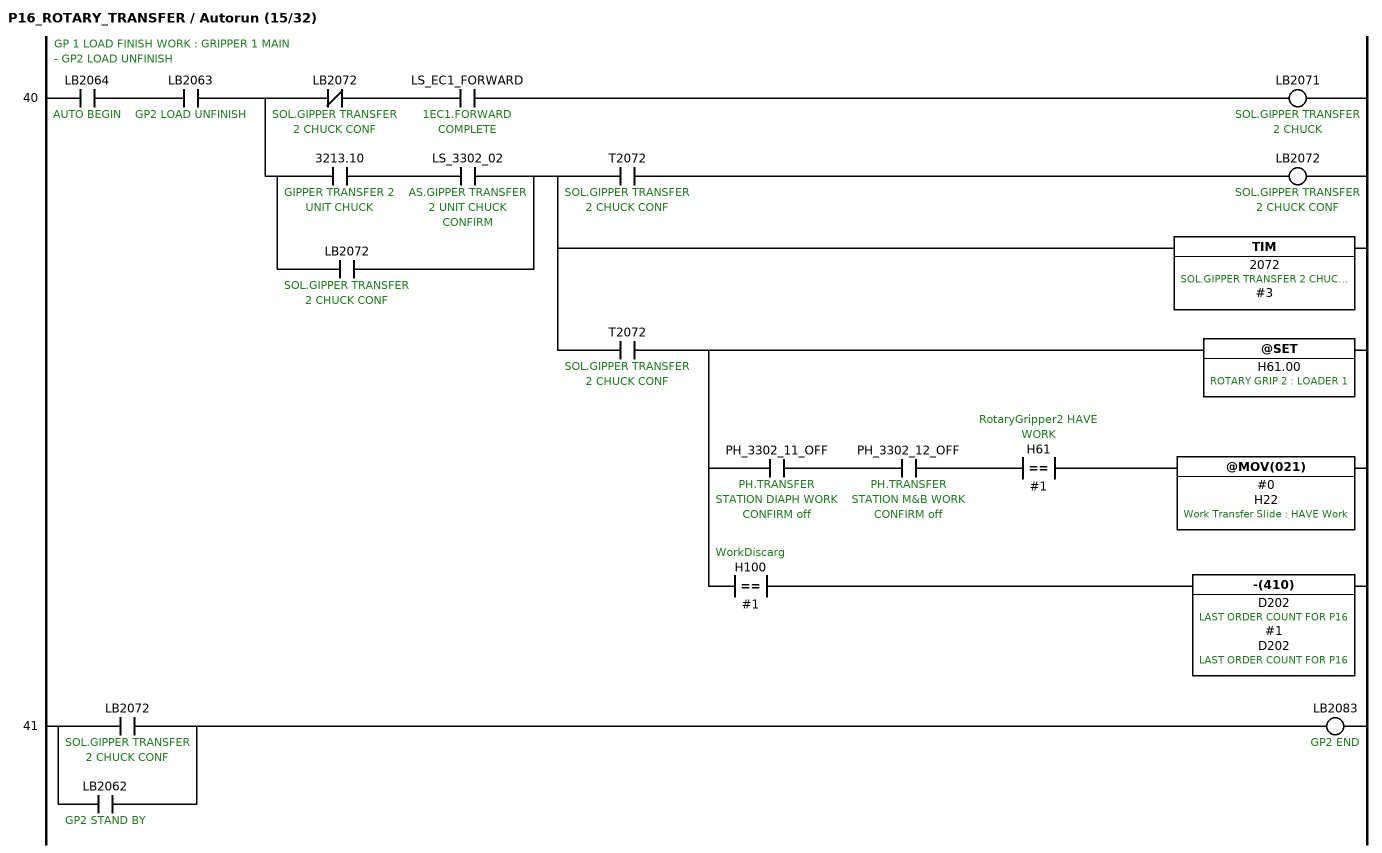
; rung 40: GP 1 LOAD FINISH WORK : GRIPPER 1 MAIN / - GP2 LOAD UNFINISH
LD LB2064  ; AUTO BEGIN
AND LB2063  ; GP2 LOAD UNFINISH
OUT TR0
ANDNOT LB2072  ; SOL.GIPPER TRANSFER 2 CHUCK CONF
AND LS_EC1_FORWARD  ; 1EC1.FORWARD COMPLETE
OUT LB2071  ; SOL.GIPPER TRANSFER 2 CHUCK
LD TR0
LD 3213.10  ; GIPPER TRANSFER 2 UNIT CHUCK
AND LS_3302_02  ; AS.GIPPER TRANSFER 2 UNIT CHUCK CONFIRM
OR LB2072  ; SOL.GIPPER TRANSFER 2 CHUCK CONF
ANDLD
OUT TR0
AND T2072  ; SOL.GIPPER TRANSFER 2 CHUCK CONF
OUT LB2072  ; SOL.GIPPER TRANSFER 2 CHUCK CONF
LD TR0
TIM 2072 #3  ; SOL.GIPPER TRANSFER 2 CHUCK CONF
AND T2072  ; SOL.GIPPER TRANSFER 2 CHUCK CONF
OUT TR0
@SET H61.00  ; ROTARY GRIP 2 : LOADER 1
AND PH_3302_11_OFF  ; PH.TRANSFER STATION DIAPH WORK CONFIRM off
AND PH_3302_12_OFF  ; PH.TRANSFER STATION M&B WORK CONFIRM off
AND=(300) H61 #1  ; RotaryGripper2 HAVE WORK
@MOV(021) #0 H22  ; Work Transfer Slide : HAVE Work
LD TR0
AND=(300) H100 #1  ; WorkDiscarg
-(410) D202 #1 D202  ; LAST ORDER COUNT FOR P16
; rung 41
LD LB2072  ; SOL.GIPPER TRANSFER 2 CHUCK CONF
OR LB2062  ; GP2 STAND BY
OUT LB2083  ; GP2 END

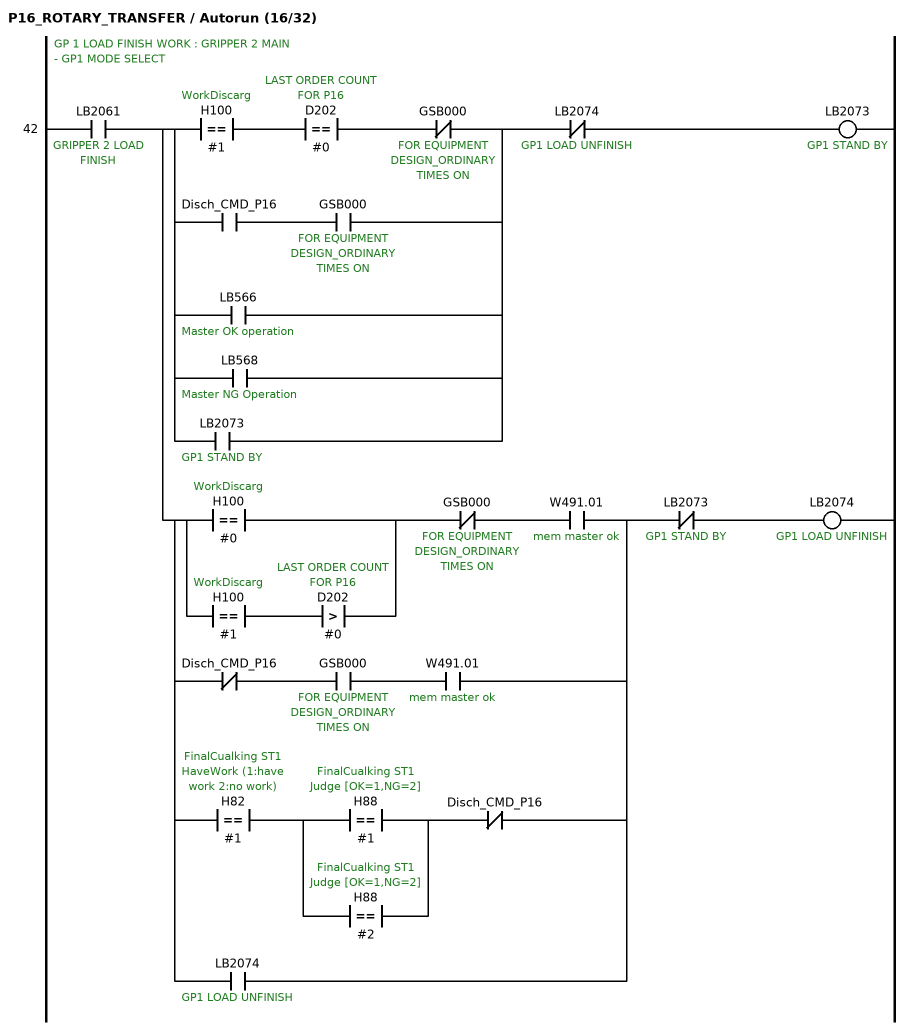
; rung 42: GP 1 LOAD FINISH WORK : GRIPPER 2 MAIN / - GP1 MODE SELECT
LD LB2061  ; GRIPPER 2 LOAD FINISH
OUT TR0
LD=(300) H100 #1  ; WorkDiscarg
AND=(300) D202 #0  ; LAST ORDER COUNT FOR P16
ANDNOT GSB000  ; FOR EQUIPMENT DESIGN_ORDINARY TIMES ON
LD Disch_CMD_P16
AND GSB000  ; FOR EQUIPMENT DESIGN_ORDINARY TIMES ON
ORLD
OR LB566  ; Master OK operation
OR LB568  ; Master NG Operation
OR LB2073  ; GP1 STAND BY
ANDLD
ANDNOT LB2074  ; GP1 LOAD UNFINISH
OUT LB2073  ; GP1 STAND BY
LD TR0
LD=(300) H100 #0  ; WorkDiscarg
LD=(300) H100 #1  ; WorkDiscarg
AND>(320) D202 #0  ; LAST ORDER COUNT FOR P16
ORLD
ANDNOT GSB000  ; FOR EQUIPMENT DESIGN_ORDINARY TIMES ON
AND W491.01  ; mem master ok
LDNOT Disch_CMD_P16
AND GSB000  ; FOR EQUIPMENT DESIGN_ORDINARY TIMES ON
AND W491.01  ; mem master ok
ORLD
LD=(300) H82 #1  ; FinalCualking ST1 HaveWork (1:have work 2:no work)
LD=(300) H88 #1  ; FinalCualking ST1 Judge [OK=1,NG=2]
OR=(300) H88 #2  ; FinalCualking ST1 Judge [OK=1,NG=2]
ANDLD
ANDNOT Disch_CMD_P16
ORLD
OR LB2074  ; GP1 LOAD UNFINISH
ANDLD
ANDNOT LB2073  ; GP1 STAND BY
OUT LB2074  ; GP1 LOAD UNFINISH

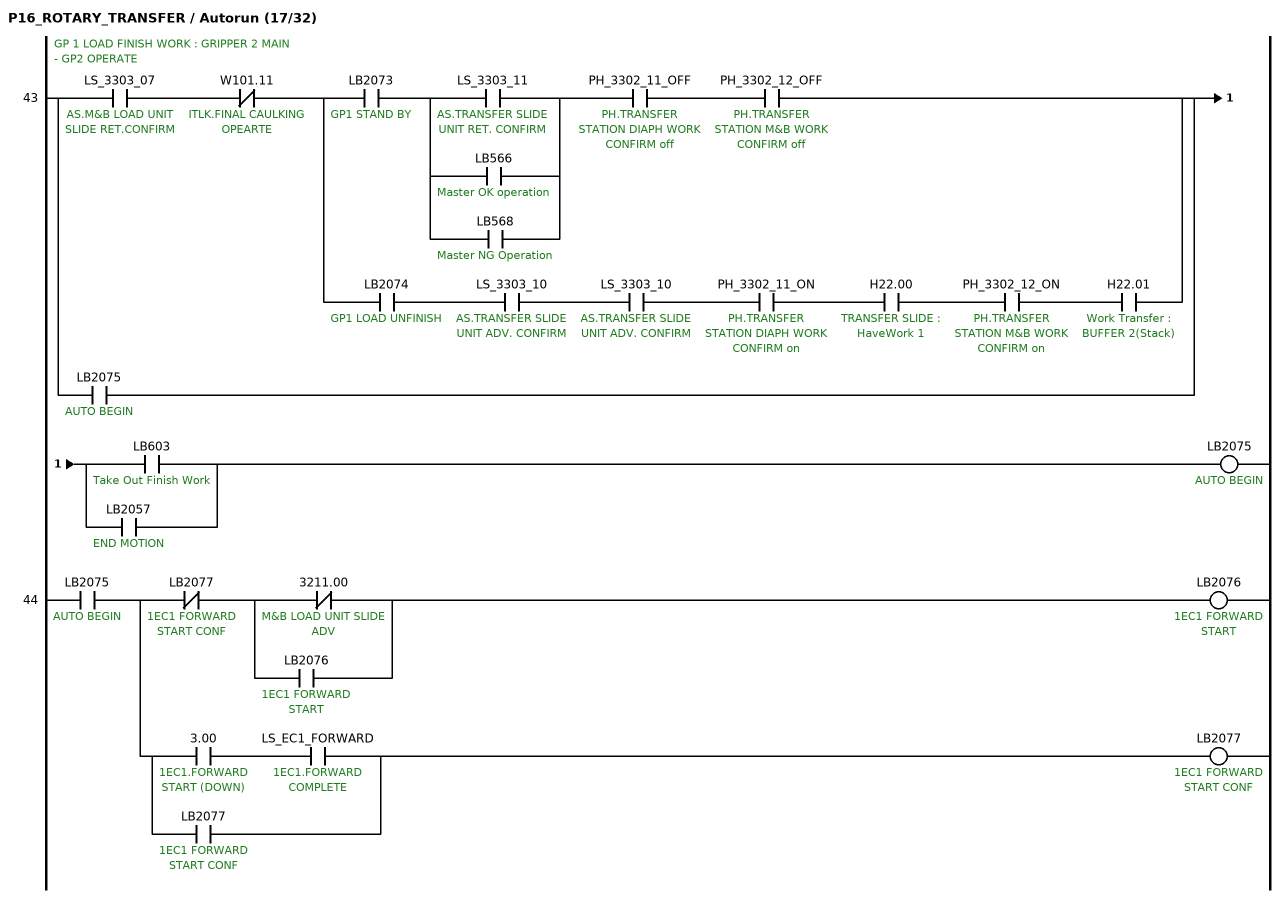
; rung 43: GP 1 LOAD FINISH WORK : GRIPPER 2 MAIN / - GP2 OPERATE
LD LS_3303_07  ; AS.M&B LOAD UNIT SLIDE RET.CONFIRM
ANDNOT W101.11  ; ITLK.FINAL CAULKING OPEARTE
LD LB2073  ; GP1 STAND BY
LD LS_3303_11  ; AS.TRANSFER SLIDE UNIT RET. CONFIRM
OR LB566  ; Master OK operation
OR LB568  ; Master NG Operation
ANDLD
AND PH_3302_11_OFF  ; PH.TRANSFER STATION DIAPH WORK CONFIRM off
AND PH_3302_12_OFF  ; PH.TRANSFER STATION M&B WORK CONFIRM off
LD LB2074  ; GP1 LOAD UNFINISH
AND LS_3303_10  ; AS.TRANSFER SLIDE UNIT ADV. CONFIRM
AND LS_3303_10  ; AS.TRANSFER SLIDE UNIT ADV. CONFIRM
AND PH_3302_11_ON  ; PH.TRANSFER STATION DIAPH WORK CONFIRM on
AND H22.00  ; TRANSFER SLIDE : HaveWork 1
AND PH_3302_12_ON  ; PH.TRANSFER STATION M&B WORK CONFIRM on
AND H22.01  ; Work Transfer : BUFFER 2(Stack)
ORLD
ANDLD
OR LB2075  ; AUTO BEGIN
LD LB603  ; Take Out Finish Work
OR LB2057  ; END MOTION
ANDLD
OUT LB2075  ; AUTO BEGIN
; rung 44
LD LB2075  ; AUTO BEGIN
OUT TR0
ANDNOT LB2077  ; 1EC1 FORWARD START CONF
LDNOT 3211.00  ; M&B LOAD UNIT SLIDE ADV
OR LB2076  ; 1EC1 FORWARD START
ANDLD
OUT LB2076  ; 1EC1 FORWARD START
LD TR0
LD 3.00  ; 1EC1.FORWARD START (DOWN)
AND LS_EC1_FORWARD  ; 1EC1.FORWARD COMPLETE
OR LB2077  ; 1EC1 FORWARD START CONF
ANDLD
OUT LB2077  ; 1EC1 FORWARD START CONF

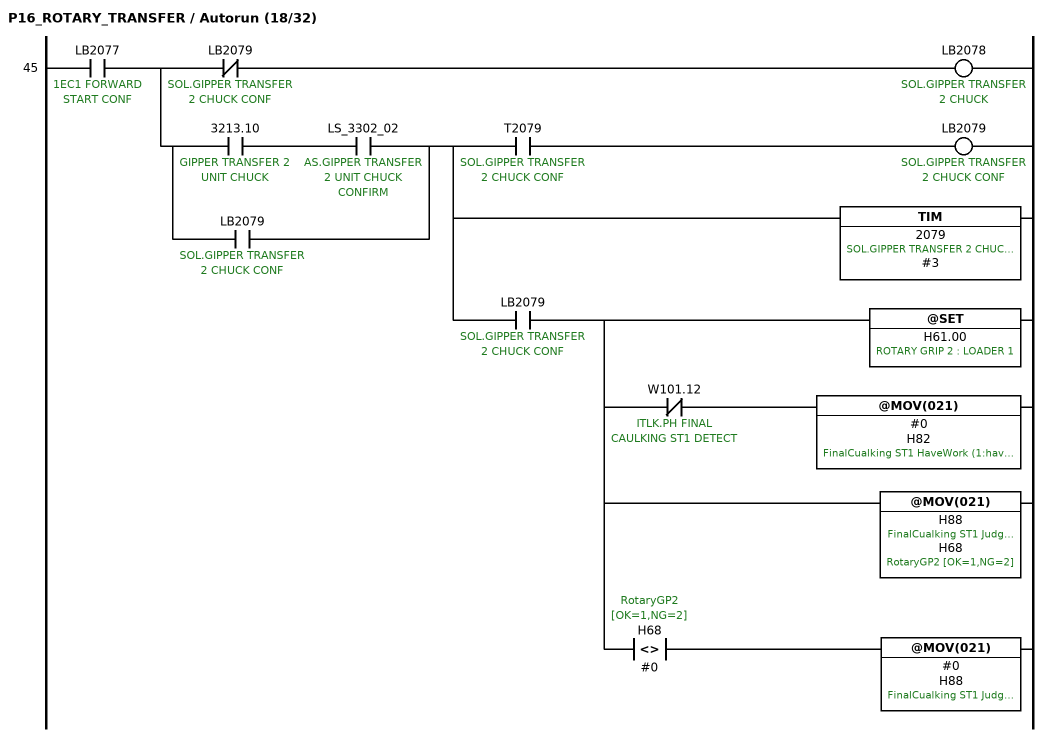
; rung 45
LD LB2077  ; 1EC1 FORWARD START CONF
OUT TR0
ANDNOT LB2079  ; SOL.GIPPER TRANSFER 2 CHUCK CONF
OUT LB2078  ; SOL.GIPPER TRANSFER 2 CHUCK
LD TR0
LD 3213.10  ; GIPPER TRANSFER 2 UNIT CHUCK
AND LS_3302_02  ; AS.GIPPER TRANSFER 2 UNIT CHUCK CONFIRM
OR LB2079  ; SOL.GIPPER TRANSFER 2 CHUCK CONF
ANDLD
OUT TR0
AND T2079  ; SOL.GIPPER TRANSFER 2 CHUCK CONF
OUT LB2079  ; SOL.GIPPER TRANSFER 2 CHUCK CONF
LD TR0
TIM 2079 #3  ; SOL.GIPPER TRANSFER 2 CHUCK CONF
AND LB2079  ; SOL.GIPPER TRANSFER 2 CHUCK CONF
OUT TR0
@SET H61.00  ; ROTARY GRIP 2 : LOADER 1
ANDNOT W101.12  ; ITLK.PH FINAL CAULKING ST1 DETECT
@MOV(021) #0 H82  ; FinalCualking ST1 HaveWork (1:have work 2:no work)
LD TR0
@MOV(021) H88 H68  ; FinalCualking ST1 Judge [OK=1,NG=2], RotaryGP2 [OK=1,NG=2]
AND<>(305) H68 #0  ; RotaryGP2 [OK=1,NG=2]
@MOV(021) #0 H88  ; FinalCualking ST1 Judge [OK=1,NG=2]

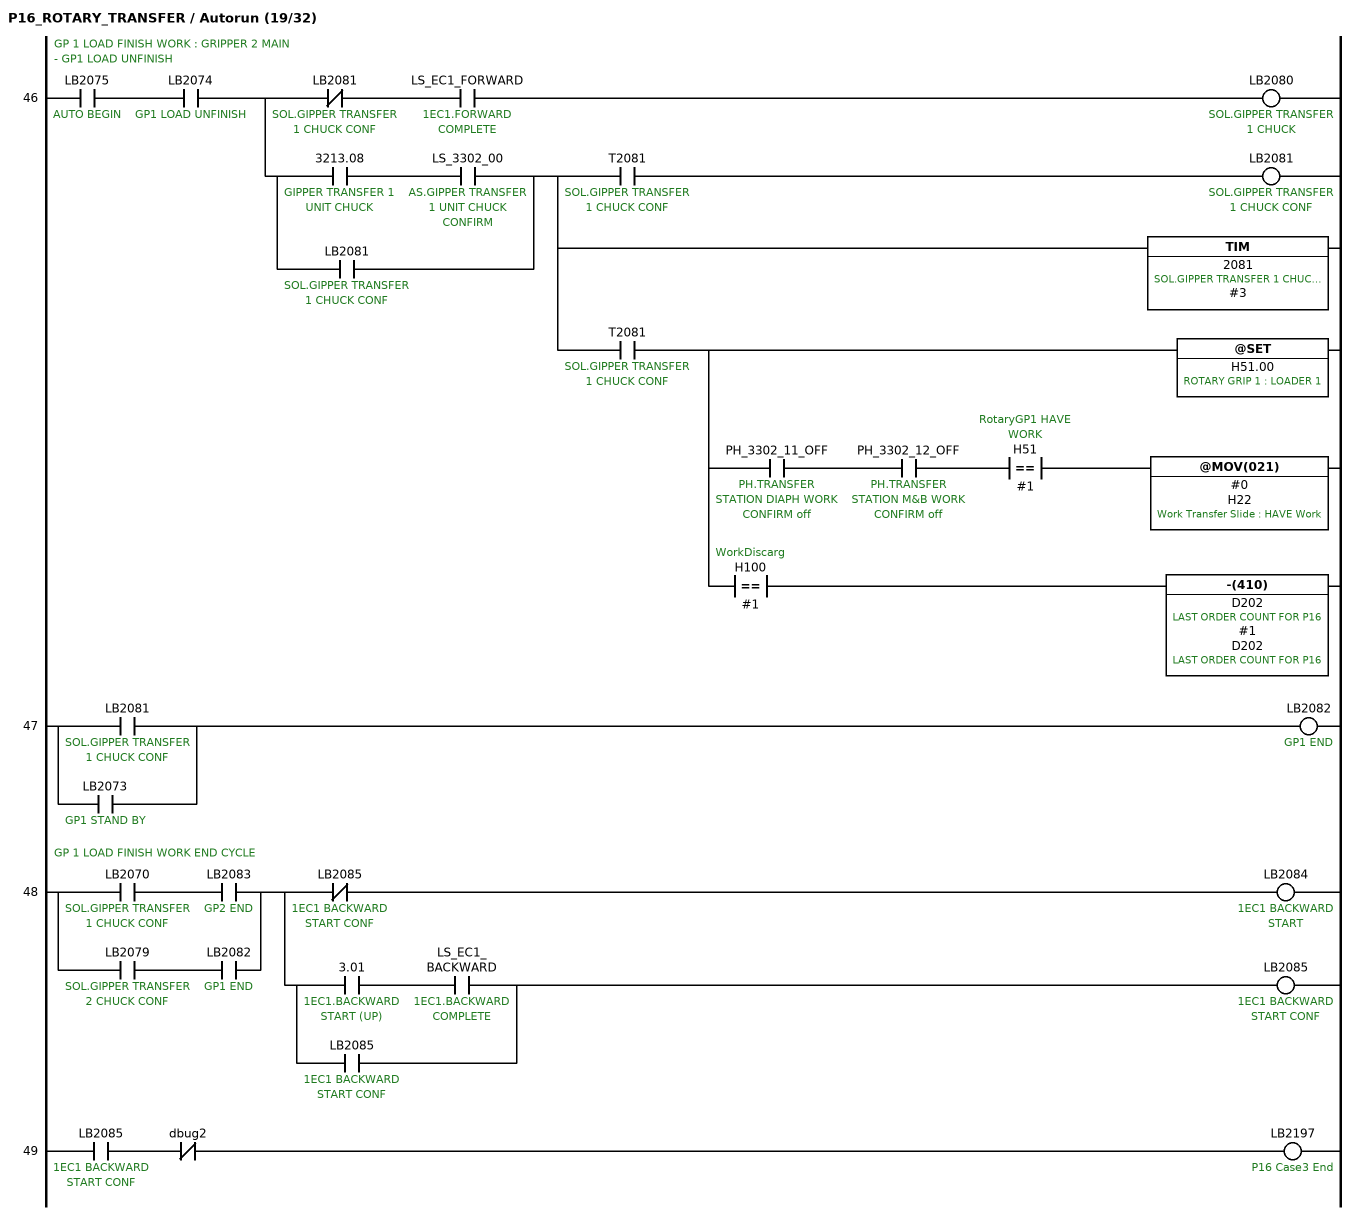
; rung 46: GP 1 LOAD FINISH WORK : GRIPPER 2 MAIN / - GP1 LOAD UNFINISH
LD LB2075  ; AUTO BEGIN
AND LB2074  ; GP1 LOAD UNFINISH
OUT TR0
ANDNOT LB2081  ; SOL.GIPPER TRANSFER 1 CHUCK CONF
AND LS_EC1_FORWARD  ; 1EC1.FORWARD COMPLETE
OUT LB2080  ; SOL.GIPPER TRANSFER 1 CHUCK
LD TR0
LD 3213.08  ; GIPPER TRANSFER 1 UNIT CHUCK
AND LS_3302_00  ; AS.GIPPER TRANSFER 1 UNIT CHUCK CONFIRM
OR LB2081  ; SOL.GIPPER TRANSFER 1 CHUCK CONF
ANDLD
OUT TR0
AND T2081  ; SOL.GIPPER TRANSFER 1 CHUCK CONF
OUT LB2081  ; SOL.GIPPER TRANSFER 1 CHUCK CONF
LD TR0
TIM 2081 #3  ; SOL.GIPPER TRANSFER 1 CHUCK CONF
AND T2081  ; SOL.GIPPER TRANSFER 1 CHUCK CONF
OUT TR0
@SET H51.00  ; ROTARY GRIP 1 : LOADER 1
AND PH_3302_11_OFF  ; PH.TRANSFER STATION DIAPH WORK CONFIRM off
AND PH_3302_12_OFF  ; PH.TRANSFER STATION M&B WORK CONFIRM off
AND=(300) H51 #1  ; RotaryGP1 HAVE WORK
@MOV(021) #0 H22  ; Work Transfer Slide : HAVE Work
LD TR0
AND=(300) H100 #1  ; WorkDiscarg
-(410) D202 #1 D202  ; LAST ORDER COUNT FOR P16
; rung 47
LD LB2081  ; SOL.GIPPER TRANSFER 1 CHUCK CONF
OR LB2073  ; GP1 STAND BY
OUT LB2082  ; GP1 END
; rung 48: GP 1 LOAD FINISH WORK END CYCLE
LD LB2070  ; SOL.GIPPER TRANSFER 1 CHUCK CONF
AND LB2083  ; GP2 END
LD LB2079  ; SOL.GIPPER TRANSFER 2 CHUCK CONF
AND LB2082  ; GP1 END
ORLD
OUT TR0
ANDNOT LB2085  ; 1EC1 BACKWARD START CONF
OUT LB2084  ; 1EC1 BACKWARD START
LD TR0
LD 3.01  ; 1EC1.BACKWARD START (UP)
AND LS_EC1_BACKWARD  ; 1EC1.BACKWARD COMPLETE
OR LB2085  ; 1EC1 BACKWARD START CONF
ANDLD
OUT LB2085  ; 1EC1 BACKWARD START CONF
; rung 49
LD LB2085  ; 1EC1 BACKWARD START CONF
ANDNOT dbug2
OUT LB2197  ; P16 Case3 End

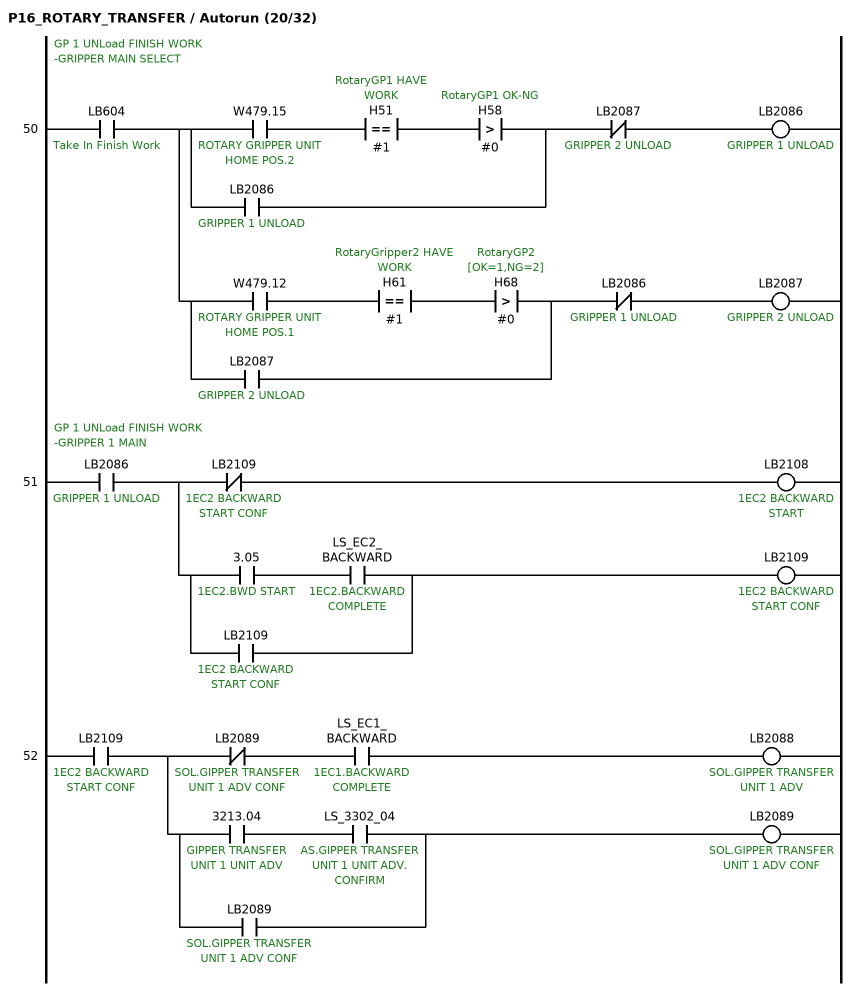
; rung 50: GP 1 UNLoad FINISH WORK / -GRIPPER MAIN SELECT
LD LB604  ; Take In Finish Work
OUT TR0
LD W479.15  ; ROTARY GRIPPER UNIT HOME POS.2
AND=(300) H51 #1  ; RotaryGP1 HAVE WORK
AND>(320) H58 #0  ; RotaryGP1 OK-NG
OR LB2086  ; GRIPPER 1 UNLOAD
ANDLD
ANDNOT LB2087  ; GRIPPER 2 UNLOAD
OUT LB2086  ; GRIPPER 1 UNLOAD
LD TR0
LD W479.12  ; ROTARY GRIPPER UNIT HOME POS.1
AND=(300) H61 #1  ; RotaryGripper2 HAVE WORK
AND>(320) H68 #0  ; RotaryGP2 [OK=1,NG=2]
OR LB2087  ; GRIPPER 2 UNLOAD
ANDLD
ANDNOT LB2086  ; GRIPPER 1 UNLOAD
OUT LB2087  ; GRIPPER 2 UNLOAD
; rung 51: GP 1 UNLoad FINISH WORK / -GRIPPER 1 MAIN
LD LB2086  ; GRIPPER 1 UNLOAD
OUT TR0
ANDNOT LB2109  ; 1EC2 BACKWARD START CONF
OUT LB2108  ; 1EC2 BACKWARD START
LD TR0
LD 3.05  ; 1EC2.BWD START
AND LS_EC2_BACKWARD  ; 1EC2.BACKWARD COMPLETE
OR LB2109  ; 1EC2 BACKWARD START CONF
ANDLD
OUT LB2109  ; 1EC2 BACKWARD START CONF
; rung 52
LD LB2109  ; 1EC2 BACKWARD START CONF
OUT TR0
ANDNOT LB2089  ; SOL.GIPPER TRANSFER UNIT 1 ADV CONF
AND LS_EC1_BACKWARD  ; 1EC1.BACKWARD COMPLETE
OUT LB2088  ; SOL.GIPPER TRANSFER UNIT 1 ADV
LD TR0
LD 3213.04  ; GIPPER TRANSFER UNIT 1 UNIT ADV
AND LS_3302_04  ; AS.GIPPER TRANSFER UNIT 1 UNIT ADV. CONFIRM
OR LB2089  ; SOL.GIPPER TRANSFER UNIT 1 ADV CONF
ANDLD
OUT LB2089  ; SOL.GIPPER TRANSFER UNIT 1 ADV CONF

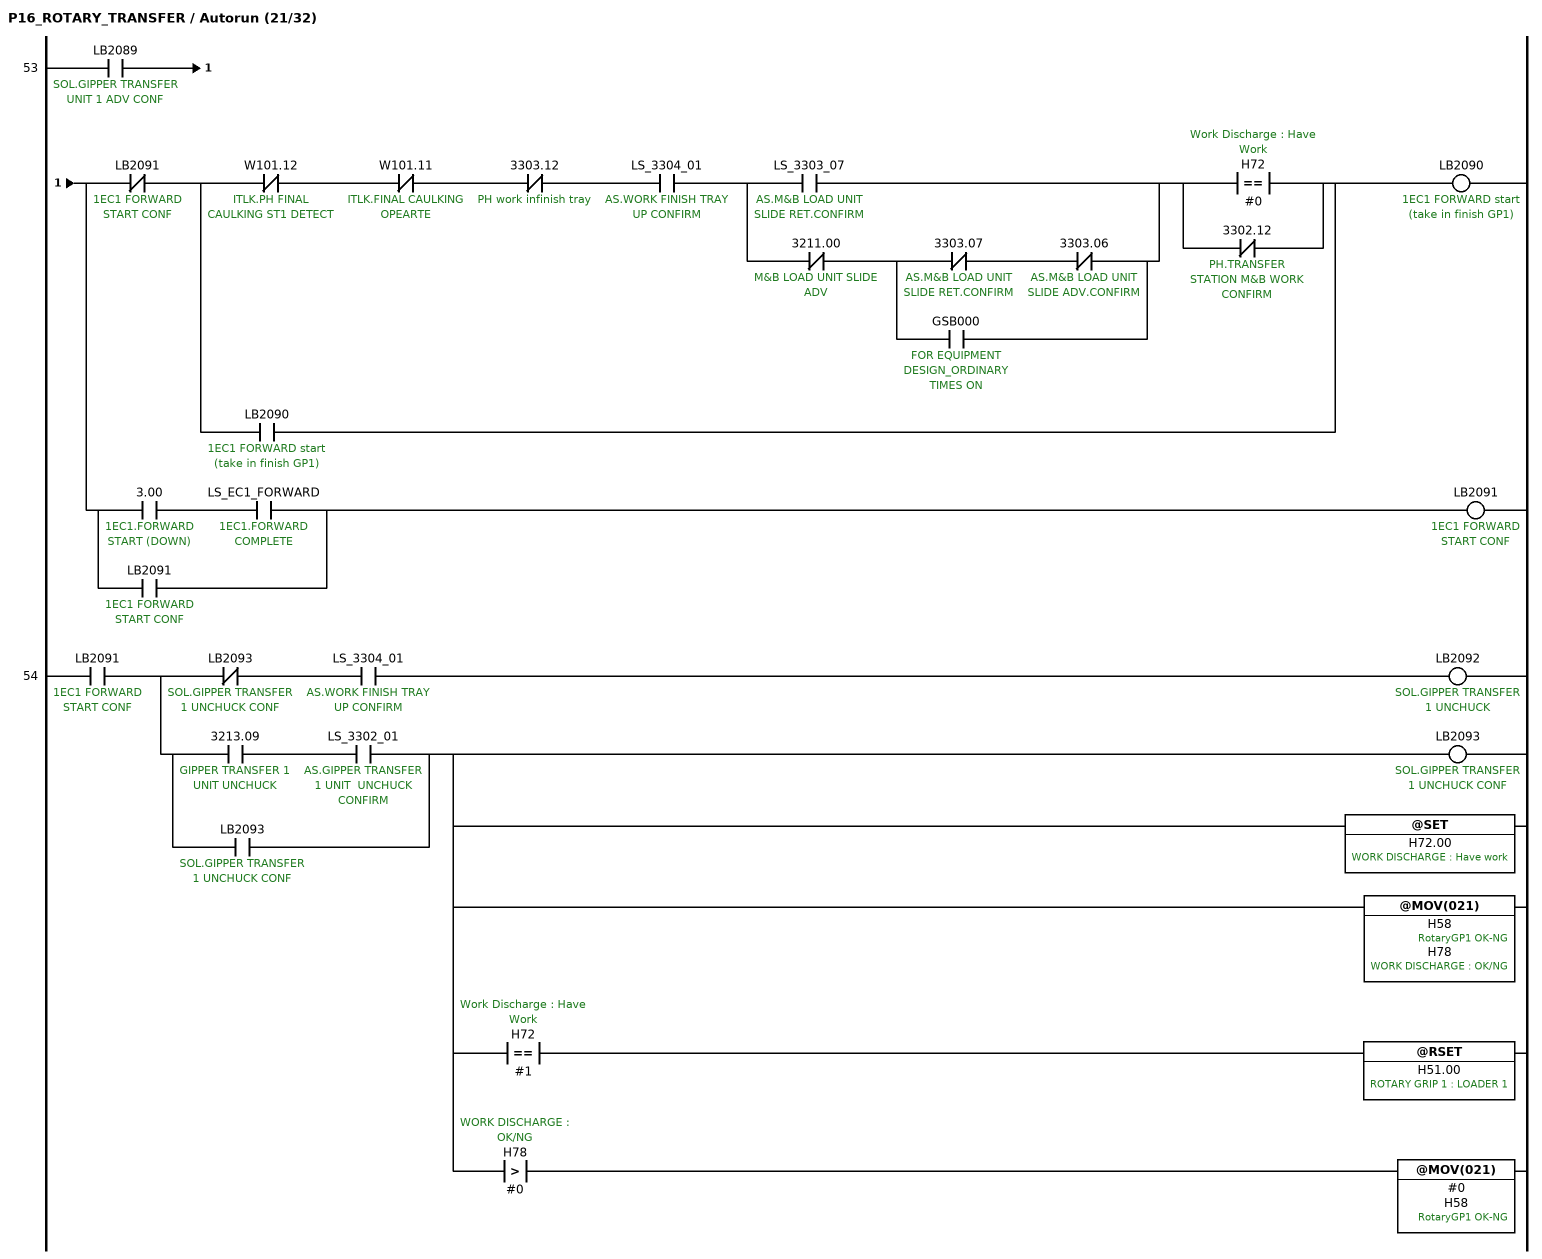
; rung 53
LD LB2089  ; SOL.GIPPER TRANSFER UNIT 1 ADV CONF
OUT TR0
ANDNOT LB2091  ; 1EC1 FORWARD START CONF
LDNOT W101.12  ; ITLK.PH FINAL CAULKING ST1 DETECT
ANDNOT W101.11  ; ITLK.FINAL CAULKING OPEARTE
ANDNOT 3303.12  ; PH work infinish tray
AND LS_3304_01  ; AS.WORK FINISH TRAY UP CONFIRM
LD LS_3303_07  ; AS.M&B LOAD UNIT SLIDE RET.CONFIRM
LDNOT 3211.00  ; M&B LOAD UNIT SLIDE ADV
LDNOT 3303.07  ; AS.M&B LOAD UNIT SLIDE RET.CONFIRM
ANDNOT 3303.06  ; AS.M&B LOAD UNIT SLIDE ADV.CONFIRM
OR GSB000  ; FOR EQUIPMENT DESIGN_ORDINARY TIMES ON
ANDLD
ORLD
ANDLD
LD=(300) H72 #0  ; Work Discharge : Have Work
ORNOT 3302.12  ; PH.TRANSFER STATION M&B WORK CONFIRM
ANDLD
OR LB2090  ; 1EC1 FORWARD start (take in finish GP1)
ANDLD
OUT LB2090  ; 1EC1 FORWARD start (take in finish GP1)
LD TR0
LD 3.00  ; 1EC1.FORWARD START (DOWN)
AND LS_EC1_FORWARD  ; 1EC1.FORWARD COMPLETE
OR LB2091  ; 1EC1 FORWARD START CONF
ANDLD
OUT LB2091  ; 1EC1 FORWARD START CONF
; rung 54
LD LB2091  ; 1EC1 FORWARD START CONF
OUT TR0
ANDNOT LB2093  ; SOL.GIPPER TRANSFER 1 UNCHUCK CONF
AND LS_3304_01  ; AS.WORK FINISH TRAY UP CONFIRM
OUT LB2092  ; SOL.GIPPER TRANSFER 1 UNCHUCK
LD TR0
LD 3213.09  ; GIPPER TRANSFER 1 UNIT UNCHUCK
AND LS_3302_01  ; AS.GIPPER TRANSFER 1 UNIT  UNCHUCK CONFIRM
OR LB2093  ; SOL.GIPPER TRANSFER 1 UNCHUCK CONF
ANDLD
OUT TR0
OUT LB2093  ; SOL.GIPPER TRANSFER 1 UNCHUCK CONF
@SET H72.00  ; WORK DISCHARGE : Have work
@MOV(021) H58 H78  ; RotaryGP1 OK-NG, WORK DISCHARGE : OK/NG
AND=(300) H72 #1  ; Work Discharge : Have Work
@RSET H51.00  ; ROTARY GRIP 1 : LOADER 1
LD TR0
AND>(320) H78 #0  ; WORK DISCHARGE : OK/NG
@MOV(021) #0 H58  ; RotaryGP1 OK-NG

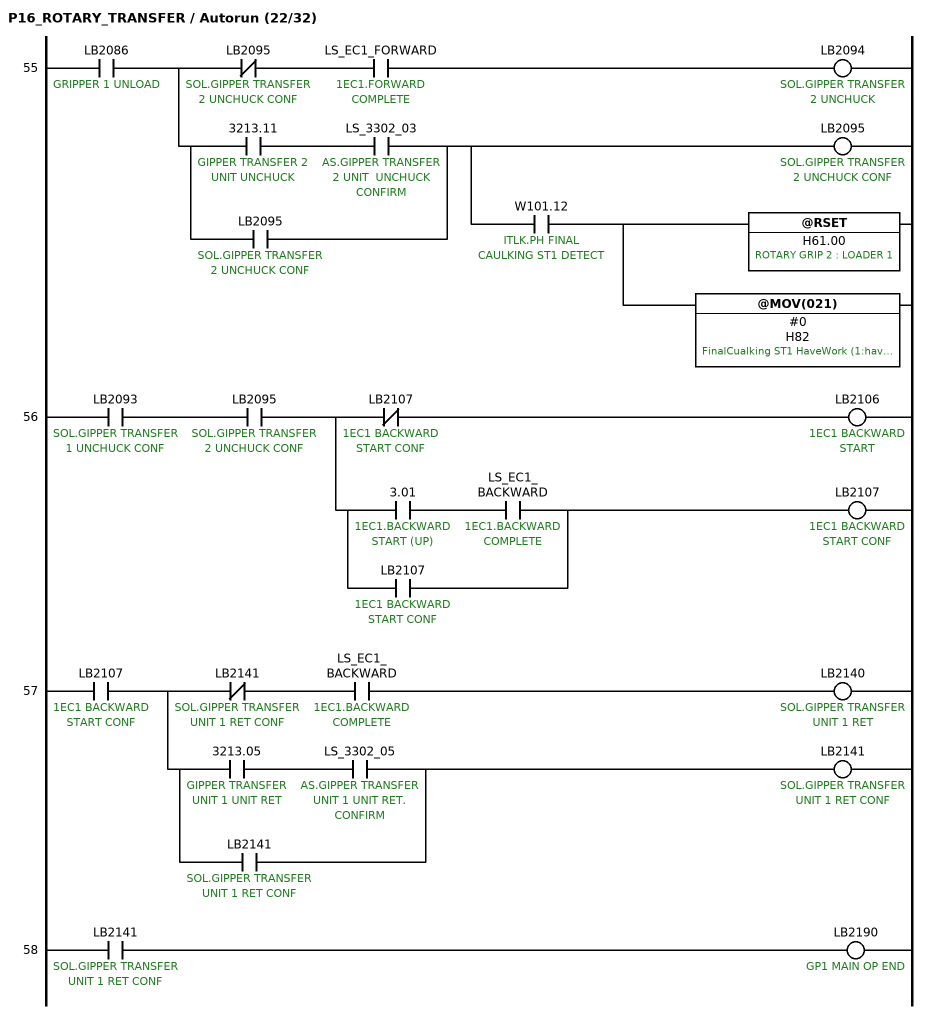
; rung 55
LD LB2086  ; GRIPPER 1 UNLOAD
OUT TR0
ANDNOT LB2095  ; SOL.GIPPER TRANSFER 2 UNCHUCK CONF
AND LS_EC1_FORWARD  ; 1EC1.FORWARD COMPLETE
OUT LB2094  ; SOL.GIPPER TRANSFER 2 UNCHUCK
LD TR0
LD 3213.11  ; GIPPER TRANSFER 2 UNIT UNCHUCK
AND LS_3302_03  ; AS.GIPPER TRANSFER 2 UNIT  UNCHUCK CONFIRM
OR LB2095  ; SOL.GIPPER TRANSFER 2 UNCHUCK CONF
ANDLD
OUT LB2095  ; SOL.GIPPER TRANSFER 2 UNCHUCK CONF
AND W101.12  ; ITLK.PH FINAL CAULKING ST1 DETECT
@RSET H61.00  ; ROTARY GRIP 2 : LOADER 1
@MOV(021) #0 H82  ; FinalCualking ST1 HaveWork (1:have work 2:no work)
; rung 56
LD LB2093  ; SOL.GIPPER TRANSFER 1 UNCHUCK CONF
AND LB2095  ; SOL.GIPPER TRANSFER 2 UNCHUCK CONF
OUT TR0
ANDNOT LB2107  ; 1EC1 BACKWARD START CONF
OUT LB2106  ; 1EC1 BACKWARD START
LD TR0
LD 3.01  ; 1EC1.BACKWARD START (UP)
AND LS_EC1_BACKWARD  ; 1EC1.BACKWARD COMPLETE
OR LB2107  ; 1EC1 BACKWARD START CONF
ANDLD
OUT LB2107  ; 1EC1 BACKWARD START CONF
; rung 57
LD LB2107  ; 1EC1 BACKWARD START CONF
OUT TR0
ANDNOT LB2141  ; SOL.GIPPER TRANSFER UNIT 1 RET CONF
AND LS_EC1_BACKWARD  ; 1EC1.BACKWARD COMPLETE
OUT LB2140  ; SOL.GIPPER TRANSFER UNIT 1 RET
LD TR0
LD 3213.05  ; GIPPER TRANSFER UNIT 1 UNIT RET
AND LS_3302_05  ; AS.GIPPER TRANSFER UNIT 1 UNIT RET. CONFIRM
OR LB2141  ; SOL.GIPPER TRANSFER UNIT 1 RET CONF
ANDLD
OUT LB2141  ; SOL.GIPPER TRANSFER UNIT 1 RET CONF
; rung 58
LD LB2141  ; SOL.GIPPER TRANSFER UNIT 1 RET CONF
OUT LB2190  ; GP1 MAIN OP END

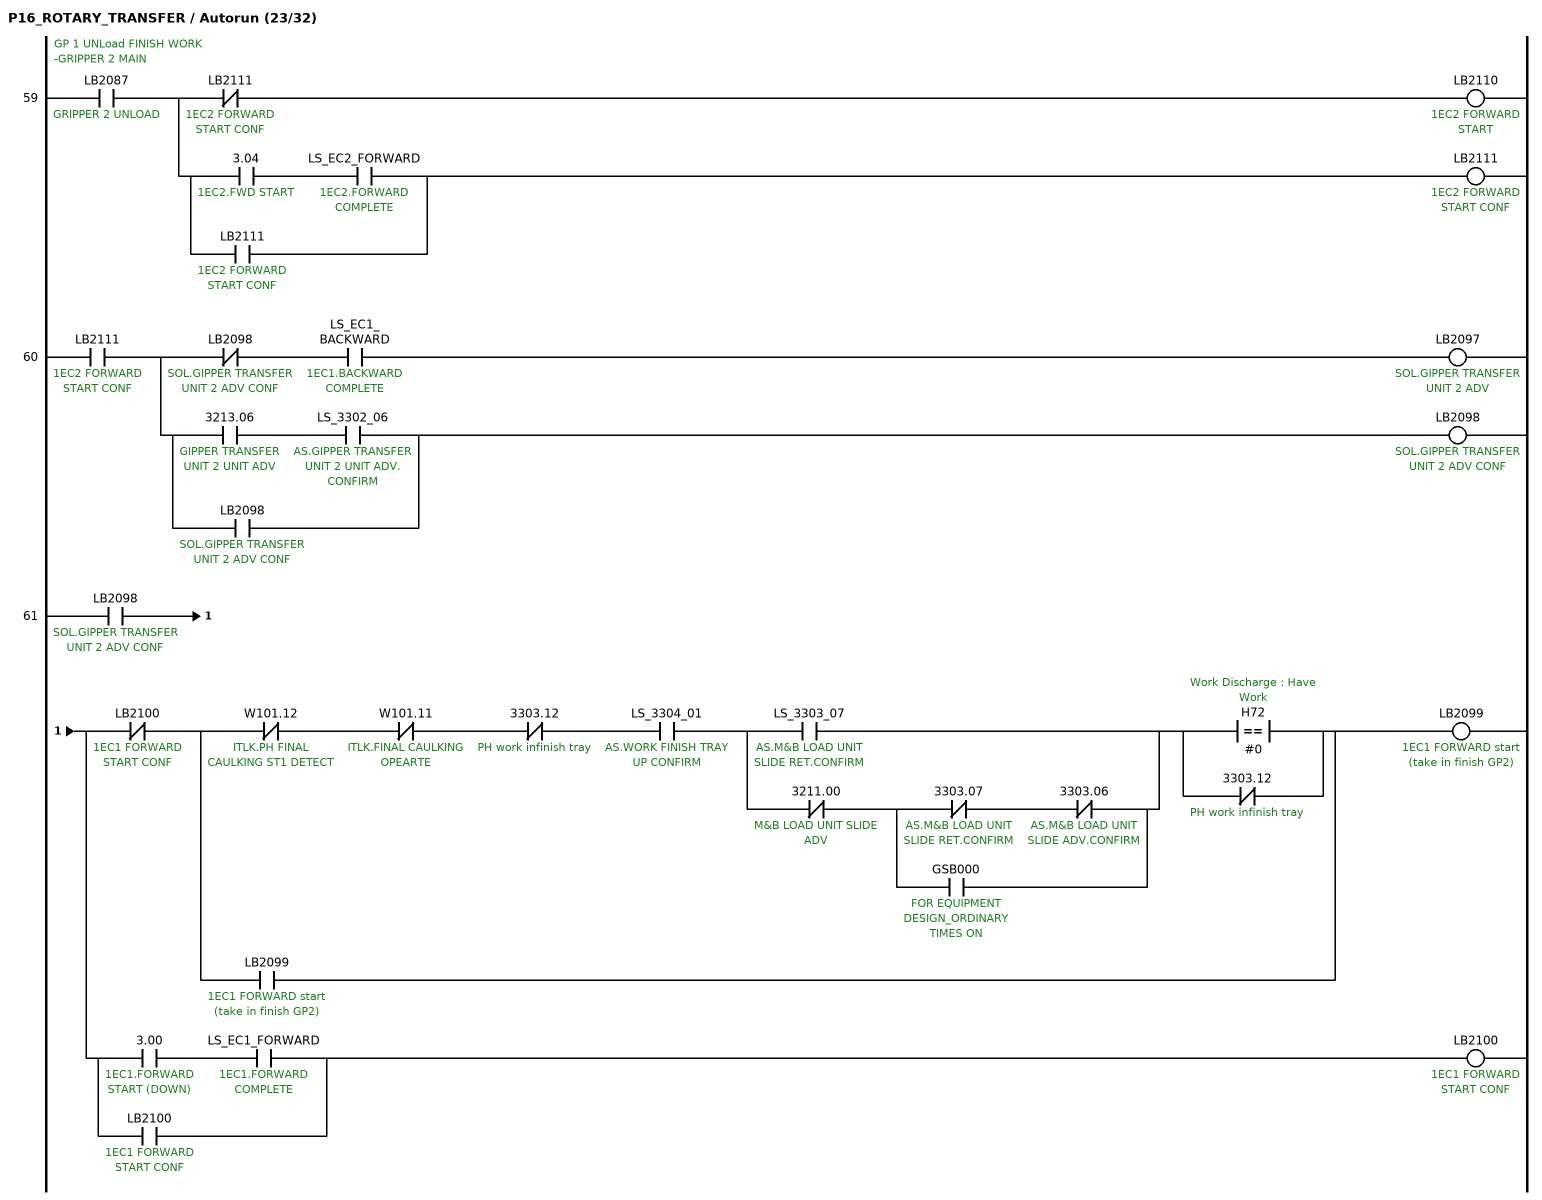
; rung 59: GP 1 UNLoad FINISH WORK / -GRIPPER 2 MAIN
LD LB2087  ; GRIPPER 2 UNLOAD
OUT TR0
ANDNOT LB2111  ; 1EC2 FORWARD START CONF
OUT LB2110  ; 1EC2 FORWARD START
LD TR0
LD 3.04  ; 1EC2.FWD START
AND LS_EC2_FORWARD  ; 1EC2.FORWARD COMPLETE
OR LB2111  ; 1EC2 FORWARD START CONF
ANDLD
OUT LB2111  ; 1EC2 FORWARD START CONF
; rung 60
LD LB2111  ; 1EC2 FORWARD START CONF
OUT TR0
ANDNOT LB2098  ; SOL.GIPPER TRANSFER UNIT 2 ADV CONF
AND LS_EC1_BACKWARD  ; 1EC1.BACKWARD COMPLETE
OUT LB2097  ; SOL.GIPPER TRANSFER UNIT 2 ADV
LD TR0
LD 3213.06  ; GIPPER TRANSFER UNIT 2 UNIT ADV
AND LS_3302_06  ; AS.GIPPER TRANSFER UNIT 2 UNIT ADV. CONFIRM
OR LB2098  ; SOL.GIPPER TRANSFER UNIT 2 ADV CONF
ANDLD
OUT LB2098  ; SOL.GIPPER TRANSFER UNIT 2 ADV CONF
; rung 61
LD LB2098  ; SOL.GIPPER TRANSFER UNIT 2 ADV CONF
OUT TR0
ANDNOT LB2100  ; 1EC1 FORWARD START CONF
LDNOT W101.12  ; ITLK.PH FINAL CAULKING ST1 DETECT
ANDNOT W101.11  ; ITLK.FINAL CAULKING OPEARTE
ANDNOT 3303.12  ; PH work infinish tray
AND LS_3304_01  ; AS.WORK FINISH TRAY UP CONFIRM
LD LS_3303_07  ; AS.M&B LOAD UNIT SLIDE RET.CONFIRM
LDNOT 3211.00  ; M&B LOAD UNIT SLIDE ADV
LDNOT 3303.07  ; AS.M&B LOAD UNIT SLIDE RET.CONFIRM
ANDNOT 3303.06  ; AS.M&B LOAD UNIT SLIDE ADV.CONFIRM
OR GSB000  ; FOR EQUIPMENT DESIGN_ORDINARY TIMES ON
ANDLD
ORLD
ANDLD
LD=(300) H72 #0  ; Work Discharge : Have Work
ORNOT 3303.12  ; PH work infinish tray
ANDLD
OR LB2099  ; 1EC1 FORWARD start (take in finish GP2)
ANDLD
OUT LB2099  ; 1EC1 FORWARD start (take in finish GP2)
LD TR0
LD 3.00  ; 1EC1.FORWARD START (DOWN)
AND LS_EC1_FORWARD  ; 1EC1.FORWARD COMPLETE
OR LB2100  ; 1EC1 FORWARD START CONF
ANDLD
OUT LB2100  ; 1EC1 FORWARD START CONF

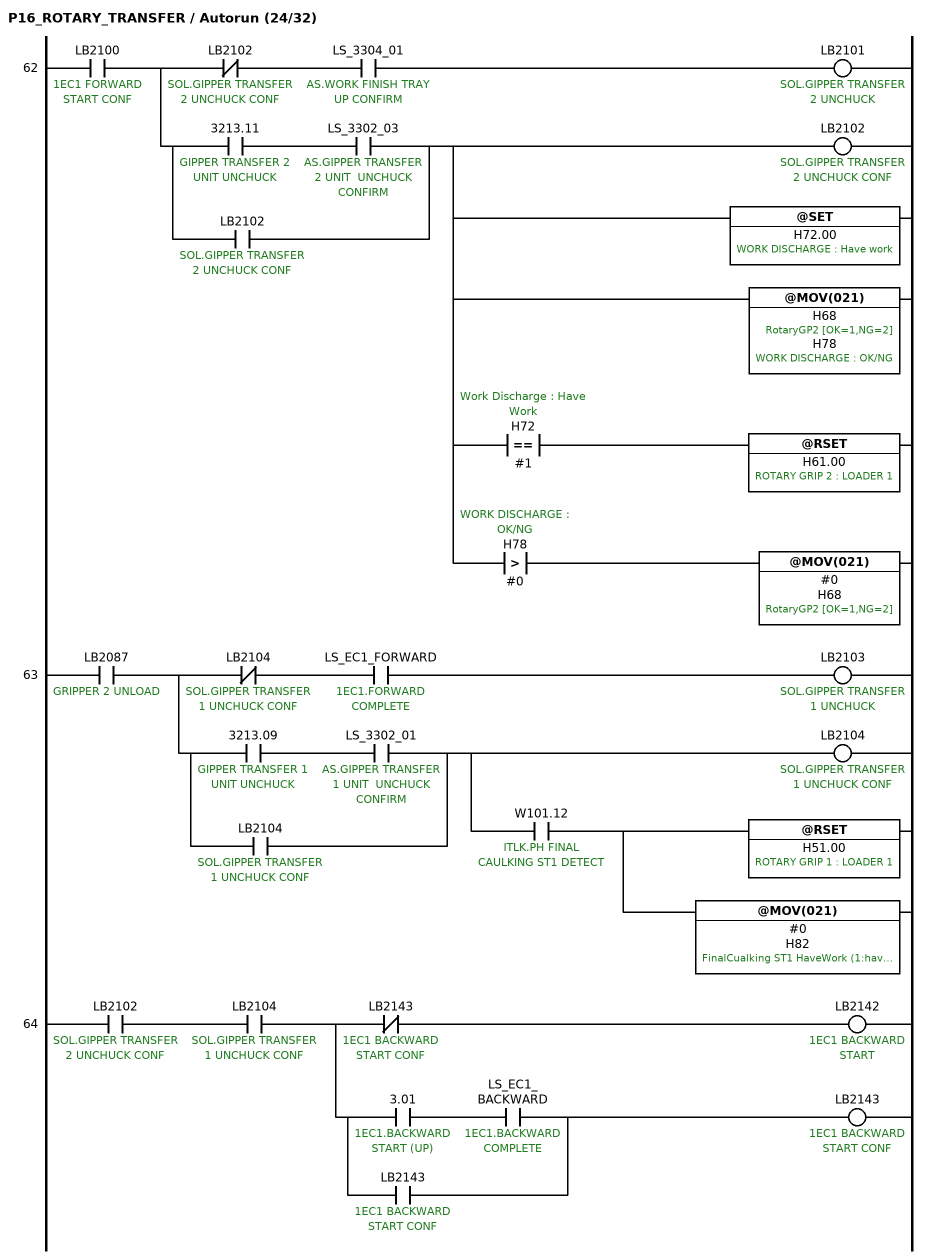
; rung 62
LD LB2100  ; 1EC1 FORWARD START CONF
OUT TR0
ANDNOT LB2102  ; SOL.GIPPER TRANSFER 2 UNCHUCK CONF
AND LS_3304_01  ; AS.WORK FINISH TRAY UP CONFIRM
OUT LB2101  ; SOL.GIPPER TRANSFER 2 UNCHUCK
LD TR0
LD 3213.11  ; GIPPER TRANSFER 2 UNIT UNCHUCK
AND LS_3302_03  ; AS.GIPPER TRANSFER 2 UNIT  UNCHUCK CONFIRM
OR LB2102  ; SOL.GIPPER TRANSFER 2 UNCHUCK CONF
ANDLD
OUT TR0
OUT LB2102  ; SOL.GIPPER TRANSFER 2 UNCHUCK CONF
@SET H72.00  ; WORK DISCHARGE : Have work
@MOV(021) H68 H78  ; RotaryGP2 [OK=1,NG=2], WORK DISCHARGE : OK/NG
AND=(300) H72 #1  ; Work Discharge : Have Work
@RSET H61.00  ; ROTARY GRIP 2 : LOADER 1
LD TR0
AND>(320) H78 #0  ; WORK DISCHARGE : OK/NG
@MOV(021) #0 H68  ; RotaryGP2 [OK=1,NG=2]
; rung 63
LD LB2087  ; GRIPPER 2 UNLOAD
OUT TR0
ANDNOT LB2104  ; SOL.GIPPER TRANSFER 1 UNCHUCK CONF
AND LS_EC1_FORWARD  ; 1EC1.FORWARD COMPLETE
OUT LB2103  ; SOL.GIPPER TRANSFER 1 UNCHUCK
LD TR0
LD 3213.09  ; GIPPER TRANSFER 1 UNIT UNCHUCK
AND LS_3302_01  ; AS.GIPPER TRANSFER 1 UNIT  UNCHUCK CONFIRM
OR LB2104  ; SOL.GIPPER TRANSFER 1 UNCHUCK CONF
ANDLD
OUT LB2104  ; SOL.GIPPER TRANSFER 1 UNCHUCK CONF
AND W101.12  ; ITLK.PH FINAL CAULKING ST1 DETECT
@RSET H51.00  ; ROTARY GRIP 1 : LOADER 1
@MOV(021) #0 H82  ; FinalCualking ST1 HaveWork (1:have work 2:no work)
; rung 64
LD LB2102  ; SOL.GIPPER TRANSFER 2 UNCHUCK CONF
AND LB2104  ; SOL.GIPPER TRANSFER 1 UNCHUCK CONF
OUT TR0
ANDNOT LB2143  ; 1EC1 BACKWARD START CONF
OUT LB2142  ; 1EC1 BACKWARD START
LD TR0
LD 3.01  ; 1EC1.BACKWARD START (UP)
AND LS_EC1_BACKWARD  ; 1EC1.BACKWARD COMPLETE
OR LB2143  ; 1EC1 BACKWARD START CONF
ANDLD
OUT LB2143  ; 1EC1 BACKWARD START CONF

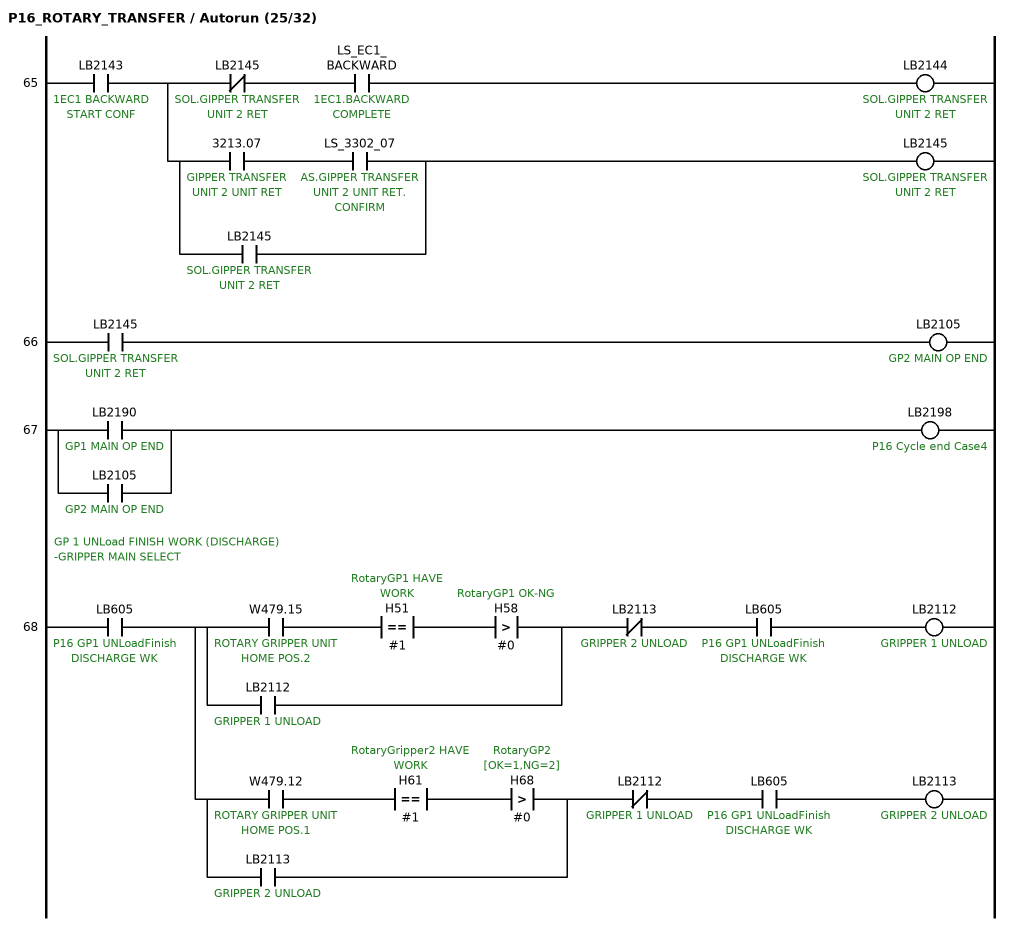
; rung 65
LD LB2143  ; 1EC1 BACKWARD START CONF
OUT TR0
ANDNOT LB2145  ; SOL.GIPPER TRANSFER UNIT 2 RET
AND LS_EC1_BACKWARD  ; 1EC1.BACKWARD COMPLETE
OUT LB2144  ; SOL.GIPPER TRANSFER UNIT 2 RET
LD TR0
LD 3213.07  ; GIPPER TRANSFER UNIT 2 UNIT RET
AND LS_3302_07  ; AS.GIPPER TRANSFER UNIT 2 UNIT RET. CONFIRM
OR LB2145  ; SOL.GIPPER TRANSFER UNIT 2 RET
ANDLD
OUT LB2145  ; SOL.GIPPER TRANSFER UNIT 2 RET
; rung 66
LD LB2145  ; SOL.GIPPER TRANSFER UNIT 2 RET
OUT LB2105  ; GP2 MAIN OP END
; rung 67
LD LB2190  ; GP1 MAIN OP END
OR LB2105  ; GP2 MAIN OP END
OUT LB2198  ; P16 Cycle end Case4
; rung 68: GP 1 UNLoad FINISH WORK (DISCHARGE) / -GRIPPER MAIN SELECT
LD LB605  ; P16 GP1 UNLoadFinish DISCHARGE WK
OUT TR0
LD W479.15  ; ROTARY GRIPPER UNIT HOME POS.2
AND=(300) H51 #1  ; RotaryGP1 HAVE WORK
AND>(320) H58 #0  ; RotaryGP1 OK-NG
OR LB2112  ; GRIPPER 1 UNLOAD
ANDLD
ANDNOT LB2113  ; GRIPPER 2 UNLOAD
AND LB605  ; P16 GP1 UNLoadFinish DISCHARGE WK
OUT LB2112  ; GRIPPER 1 UNLOAD
LD TR0
LD W479.12  ; ROTARY GRIPPER UNIT HOME POS.1
AND=(300) H61 #1  ; RotaryGripper2 HAVE WORK
AND>(320) H68 #0  ; RotaryGP2 [OK=1,NG=2]
OR LB2113  ; GRIPPER 2 UNLOAD
ANDLD
ANDNOT LB2112  ; GRIPPER 1 UNLOAD
AND LB605  ; P16 GP1 UNLoadFinish DISCHARGE WK
OUT LB2113  ; GRIPPER 2 UNLOAD

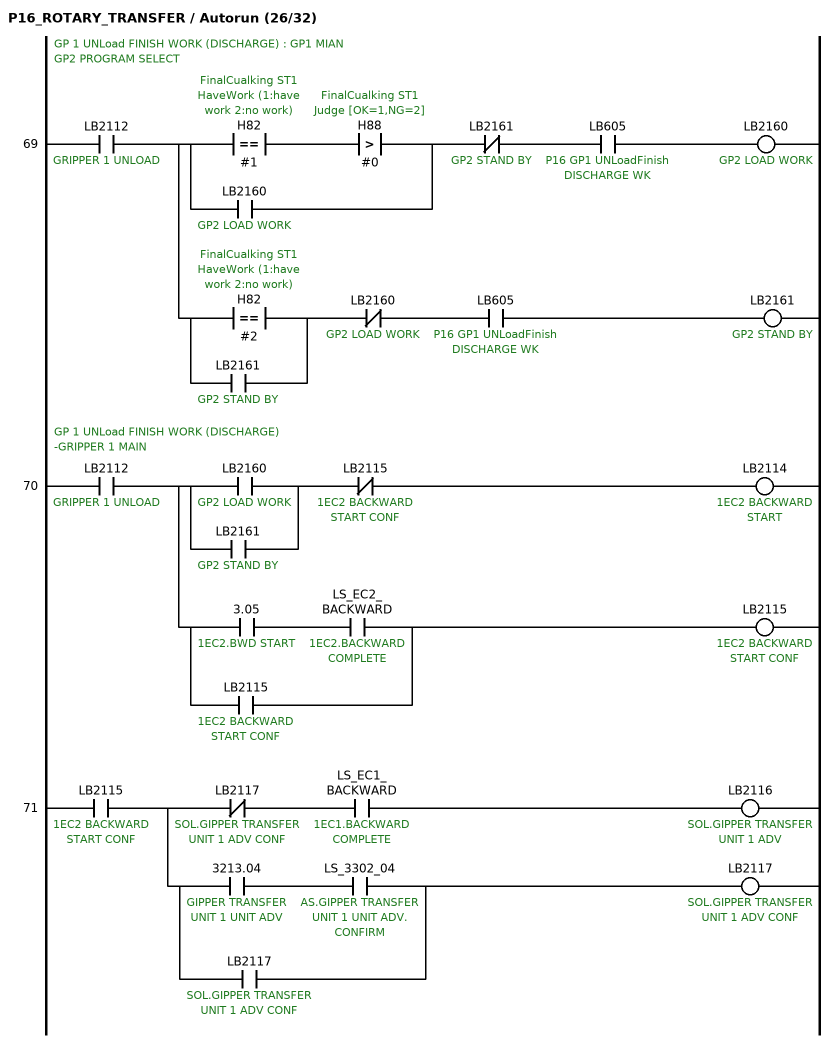
; rung 69: GP 1 UNLoad FINISH WORK (DISCHARGE) : GP1 MIAN / GP2 PROGRAM SELECT
LD LB2112  ; GRIPPER 1 UNLOAD
OUT TR0
LD=(300) H82 #1  ; FinalCualking ST1 HaveWork (1:have work 2:no work)
AND>(320) H88 #0  ; FinalCualking ST1 Judge [OK=1,NG=2]
OR LB2160  ; GP2 LOAD WORK
ANDLD
ANDNOT LB2161  ; GP2 STAND BY
AND LB605  ; P16 GP1 UNLoadFinish DISCHARGE WK
OUT LB2160  ; GP2 LOAD WORK
LD TR0
LD=(300) H82 #2  ; FinalCualking ST1 HaveWork (1:have work 2:no work)
OR LB2161  ; GP2 STAND BY
ANDLD
ANDNOT LB2160  ; GP2 LOAD WORK
AND LB605  ; P16 GP1 UNLoadFinish DISCHARGE WK
OUT LB2161  ; GP2 STAND BY
; rung 70: GP 1 UNLoad FINISH WORK (DISCHARGE) / -GRIPPER 1 MAIN
LD LB2112  ; GRIPPER 1 UNLOAD
OUT TR0
LD LB2160  ; GP2 LOAD WORK
OR LB2161  ; GP2 STAND BY
ANDLD
ANDNOT LB2115  ; 1EC2 BACKWARD START CONF
OUT LB2114  ; 1EC2 BACKWARD START
LD TR0
LD 3.05  ; 1EC2.BWD START
AND LS_EC2_BACKWARD  ; 1EC2.BACKWARD COMPLETE
OR LB2115  ; 1EC2 BACKWARD START CONF
ANDLD
OUT LB2115  ; 1EC2 BACKWARD START CONF
; rung 71
LD LB2115  ; 1EC2 BACKWARD START CONF
OUT TR0
ANDNOT LB2117  ; SOL.GIPPER TRANSFER UNIT 1 ADV CONF
AND LS_EC1_BACKWARD  ; 1EC1.BACKWARD COMPLETE
OUT LB2116  ; SOL.GIPPER TRANSFER UNIT 1 ADV
LD TR0
LD 3213.04  ; GIPPER TRANSFER UNIT 1 UNIT ADV
AND LS_3302_04  ; AS.GIPPER TRANSFER UNIT 1 UNIT ADV. CONFIRM
OR LB2117  ; SOL.GIPPER TRANSFER UNIT 1 ADV CONF
ANDLD
OUT LB2117  ; SOL.GIPPER TRANSFER UNIT 1 ADV CONF

